DATA_BLOCK "ro_steam"   // DB283
{ S7_Optimized_Access := 'FALSE' }
VERSION : 0.1
// stored: InstanceOfName ro
"ro"
BEGIN
   P[1] := 0.1;
   P[2] := 0.2;
   P[3] := 0.3;
   P[4] := 0.4;
   P[5] := 0.5;
   P[6] := 0.6;
   P[7] := 0.7;
   P[8] := 0.8;
   P[9] := 0.9;
   P[10] := 1.0;
   T[1] := 10.0;
   T[2] := 20.0;
   T[3] := 30.0;
   T[4] := 40.0;
   T[5] := 50.0;
   T[6] := 60.0;
   T[7] := 70.0;
   T[8] := 80.0;
   T[9] := 90.0;
   T[10] := 100.0;
   T[11] := 110.0;
   T[12] := 120.0;
   T[13] := 130.0;
   T[14] := 140.0;
   T[15] := 150.0;
   T[16] := 160.0;
   T[17] := 170.0;
   T[18] := 180.0;
   T[19] := 190.0;
   T[20] := 200.0;
   PT[1,1] := 1.0003;
   PT[1,2] := 1.001799;
   PT[1,3] := 1.004368;
   PT[1,4] := 1.007838;
   PT[1,5] := 1.012099;
   PT[1,6] := 1.017078;
   PT[1,7] := 1.022727;
   PT[1,8] := 1.029017;
   PT[1,9] := 1.035929;
   PT[1,10] := 1729.941;
   PT[1,11] := 1779.703;
   PT[1,12] := 1829.026;
   PT[1,13] := 1878.016;
   PT[1,14] := 1926.736;
   PT[1,15] := 1975.238;
   PT[1,16] := 2023.559;
   PT[1,17] := 2071.728;
   PT[1,18] := 2119.771;
   PT[1,19] := 2167.707;
   PT[1,20] := 2215.552;
   PT[2,1] := 1.000253;
   PT[2,2] := 1.001754;
   PT[2,3] := 1.004324;
   PT[2,4] := 1.007794;
   PT[2,5] := 1.012055;
   PT[2,6] := 1.017033;
   PT[2,7] := 1.022682;
   PT[2,8] := 1.02897;
   PT[2,9] := 1.035881;
   PT[2,10] := 1.043407;
   PT[2,11] := 1.051552;
   PT[2,12] := 903.1196;
   PT[2,13] := 928.7784;
   PT[2,14] := 954.0966;
   PT[2,15] := 979.1605;
   PT[2,16] := 1004.021;
   PT[2,17] := 1028.715;
   PT[2,18] := 1053.271;
   PT[2,19] := 1077.71;
   PT[2,20] := 1102.051;
   PT[3,1] := 1.000206;
   PT[3,2] := 1.001709;
   PT[3,3] := 1.00428;
   PT[3,4] := 1.007751;
   PT[3,5] := 1.012011;
   PT[3,6] := 1.016989;
   PT[3,7] := 1.022637;
   PT[3,8] := 1.028924;
   PT[3,9] := 1.035833;
   PT[3,10] := 1.043357;
   PT[3,11] := 1.0515;
   PT[3,12] := 1.060273;
   PT[3,13] := 1.069697;
   PT[3,14] := 629.5558;
   PT[3,15] := 646.8893;
   PT[3,16] := 663.9833;
   PT[3,17] := 680.8912;
   PT[3,18] := 697.6475;
   PT[3,19] := 714.2781;
   PT[3,20] := 730.8032;
   PT[4,1] := 1.00016;
   PT[4,2] := 1.001664;
   PT[4,3] := 1.004236;
   PT[4,4] := 1.007707;
   PT[4,5] := 1.011968;
   PT[4,6] := 1.016945;
   PT[4,7] := 1.022592;
   PT[4,8] := 1.028878;
   PT[4,9] := 1.035785;
   PT[4,10] := 1.043307;
   PT[4,11] := 1.051447;
   PT[4,12] := 1.060218;
   PT[4,13] := 1.069639;
   PT[4,14] := 1.07974;
   PT[4,15] := 480.5462;
   PT[4,16] := 493.8126;
   PT[4,17] := 506.8611;
   PT[4,18] := 519.7418;
   PT[4,19] := 532.4865;
   PT[4,20] := 545.118;
   PT[5,1] := 1.000113;
   PT[5,2] := 1.001619;
   PT[5,3] := 1.004193;
   PT[5,4] := 1.007664;
   PT[5,5] := 1.011924;
   PT[5,6] := 1.016901;
   PT[5,7] := 1.022547;
   PT[5,8] := 1.028831;
   PT[5,9] := 1.035737;
   PT[5,10] := 1.043257;
   PT[5,11] := 1.051395;
   PT[5,12] := 1.060163;
   PT[5,13] := 1.06958;
   PT[5,14] := 1.079678;
   PT[5,15] := 1.090495;
   PT[5,16] := 391.5747;
   PT[5,17] := 402.3437;
   PT[5,18] := 412.9209;
   PT[5,19] := 423.3495;
   PT[5,20] := 433.6568;
   PT[6,1] := 1.000066;
   PT[6,2] := 1.001574;
   PT[6,3] := 1.004149;
   PT[6,4] := 1.00762;
   PT[6,5] := 1.01188;
   PT[6,6] := 1.016857;
   PT[6,7] := 1.022502;
   PT[6,8] := 1.028785;
   PT[6,9] := 1.035689;
   PT[6,10] := 1.043207;
   PT[6,11] := 1.051343;
   PT[6,12] := 1.060107;
   PT[6,13] := 1.069522;
   PT[6,14] := 1.079616;
   PT[6,15] := 1.090429;
   PT[6,16] := 323.2793;
   PT[6,17] := 332.5752;
   PT[6,18] := 341.6396;
   PT[6,19] := 350.5385;
   PT[6,20] := 359.3066;
   PT[7,1] := 1.000019;
   PT[7,2] := 1.001529;
   PT[7,3] := 1.004105;
   PT[7,4] := 1.007577;
   PT[7,5] := 1.011837;
   PT[7,6] := 1.016812;
   PT[7,7] := 1.022457;
   PT[7,8] := 1.028738;
   PT[7,9] := 1.035641;
   PT[7,10] := 1.043157;
   PT[7,11] := 1.05129;
   PT[7,12] := 1.060052;
   PT[7,13] := 1.069464;
   PT[7,14] := 1.079554;
   PT[7,15] := 1.090363;
   PT[7,16] := 1.101939;
   PT[7,17] := 282.652;
   PT[7,18] := 290.6629;
   PT[7,19] := 298.4836;
   PT[7,20] := 306.162;
   PT[8,1] := 0.9999723;
   PT[8,2] := 1.001484;
   PT[8,3] := 1.004061;
   PT[8,4] := 1.007533;
   PT[8,5] := 1.011793;
   PT[8,6] := 1.016768;
   PT[8,7] := 1.022411;
   PT[8,8] := 1.028692;
   PT[8,9] := 1.035593;
   PT[8,10] := 1.043107;
   PT[8,11] := 1.051238;
   PT[8,12] := 1.059997;
   PT[8,13] := 1.069406;
   PT[8,14] := 1.079492;
   PT[8,15] := 1.090296;
   PT[8,16] := 1.101868;
   PT[8,17] := 245.1154;
   PT[8,18] := 252.3714;
   PT[8,19] := 259.3993;
   PT[8,20] := 266.2699;
   PT[9,1] := 0.9999255;
   PT[9,2] := 1.001439;
   PT[9,3] := 1.004017;
   PT[9,4] := 1.00749;
   PT[9,5] := 1.011749;
   PT[9,6] := 1.016724;
   PT[9,7] := 1.022366;
   PT[9,8] := 1.028646;
   PT[9,9] := 1.035545;
   PT[9,10] := 1.043057;
   PT[9,11] := 1.051186;
   PT[9,12] := 1.059942;
   PT[9,13] := 1.069347;
   PT[9,14] := 1.07943;
   PT[9,15] := 1.09023;
   PT[9,16] := 1.101797;
   PT[9,17] := 1.114191;
   PT[9,18] := 222.5293;
   PT[9,19] := 228.9597;
   PT[9,20] := 235.2116;
   PT[10,1] := 0.9998788;
   PT[10,2] := 1.001394;
   PT[10,3] := 1.003973;
   PT[10,4] := 1.007446;
   PT[10,5] := 1.011706;
   PT[10,6] := 1.01668;
   PT[10,7] := 1.022321;
   PT[10,8] := 1.0286;
   PT[10,9] := 1.035497;
   PT[10,10] := 1.043007;
   PT[10,11] := 1.051134;
   PT[10,12] := 1.059887;
   PT[10,13] := 1.069289;
   PT[10,14] := 1.079368;
   PT[10,15] := 1.090164;
   PT[10,16] := 1.101725;
   PT[10,17] := 1.114115;
   PT[10,18] := 198.5921;
   PT[10,19] := 204.568;
   PT[10,20] := 210.3359;
END_DATA_BLOCK

DATA_BLOCK "Qs_gas"   // DB284
{ S7_Optimized_Access := 'FALSE' }
VERSION : 0.1
// stored: InstanceOfName Qs
"Qs"
BEGIN
   ro_c := 0.7024;
   Xa := 0.00642;
   Xy := 0.00217;
END_DATA_BLOCK

DATA_BLOCK "Q1_water"   // DB286
{ S7_Optimized_Access := 'FALSE' }
VERSION : 0.1
   VAR
      Calorie : Real := 8160.0;   // Калорийность
      KPD : Real := 0.89;   // КПД
      "E" : Real := 566.0;   // Энтальпия
      Value : Real;   // Расход воды
   END_VAR
BEGIN
END_DATA_BLOCK

// folder: Analog_out

DATA_BLOCK "DV_control_frequency"   // DB149
{ S7_Optimized_Access := 'FALSE' }
AUTHOR : Dmitriy_Petrov
VERSION : 0.1
// Задание для ПЧ ДВ
// stored: InstanceOfName WRITE_ANALOG_SIGNAL
"WRITE_ANALOG_SIGNAL"
BEGIN
   N_module := 14;
   N_chanel := 1;
   HL_control_signal_new := 50.0;
   HL_control_signal := 50.0;
END_DATA_BLOCK

DATA_BLOCK "DS_control_frequency"   // DB150
{ S7_Optimized_Access := 'FALSE' }
AUTHOR : Dmitriy_Petrov
VERSION : 0.1
// Задание для ПЧ ДС
// stored: InstanceOfName WRITE_ANALOG_SIGNAL
"WRITE_ANALOG_SIGNAL"
BEGIN
   N_module := 14;
   N_chanel := 2;
   HL_control_signal_new := 50.0;
   HL_control_signal := 50.0;
END_DATA_BLOCK

// folder: Analog_sensors

DATA_BLOCK "T_water_before_economizer"   // DB1
{ S7_Optimized_Access := 'FALSE' }
AUTHOR : Dmitriy_Petrov
VERSION : 0.1
// Температура питательной воды перед экономайзером (град С)
// stored: InstanceOfName READ_ANALOG_SENSOR
"READ_ANALOG_SENSOR"
BEGIN
   N_module := 1;
   N_chanel := 1;
   HL_sensor_new := 200.0;
   HL_sensor := 200.0;
END_DATA_BLOCK

DATA_BLOCK "T_water_after_economizer"   // DB2
{ S7_Optimized_Access := 'FALSE' }
AUTHOR : Dmitriy_Petrov
VERSION : 0.1
// Температура питательной воды после экономайзера (град С)
// stored: InstanceOfName READ_ANALOG_SENSOR
"READ_ANALOG_SENSOR"
BEGIN
   N_module := 1;
   N_chanel := 2;
   HL_sensor_new := 200.0;
   HL_sensor := 200.0;
END_DATA_BLOCK

DATA_BLOCK "dP_water_boiler"   // DB3
{ S7_Optimized_Access := 'FALSE' }
AUTHOR : Dmitriy_Petrov
VERSION : 0.1
// Перепад давления питательной воды на котел (кПа)
// stored: InstanceOfName READ_ANALOG_SENSOR
"READ_ANALOG_SENSOR"
BEGIN
   N_module := 1;
   N_chanel := 3;
   HL_sensor_new := 63.0;
   HL_sensor := 63.0;
END_DATA_BLOCK

DATA_BLOCK "P_water_before_regul"   // DB4
{ S7_Optimized_Access := 'FALSE' }
AUTHOR : Dmitriy_Petrov
VERSION : 0.1
// Давление питательной воды до регулятора (МПа)
// stored: InstanceOfName READ_ANALOG_SENSOR
"READ_ANALOG_SENSOR"
BEGIN
   N_module := 1;
   N_chanel := 4;
   HL_sensor_new := 25.0;
   HL_sensor := 25.0;
END_DATA_BLOCK

DATA_BLOCK "P_water_after_regul"   // DB5
{ S7_Optimized_Access := 'FALSE' }
AUTHOR : Dmitriy_Petrov
VERSION : 0.1
// Давление питательной воды после регулятора (МПа)
// stored: InstanceOfName READ_ANALOG_SENSOR
"READ_ANALOG_SENSOR"
BEGIN
   N_module := 1;
   N_chanel := 5;
   HL_sensor_new := 2.5;
   HL_sensor := 2.5;
END_DATA_BLOCK

DATA_BLOCK "dP_steam"   // DB6
{ S7_Optimized_Access := 'FALSE' }
AUTHOR : Dmitriy_Petrov
VERSION : 0.1
// Перепад давления пара в магистраль (кПа)
// stored: InstanceOfName READ_ANALOG_SENSOR
"READ_ANALOG_SENSOR"
BEGIN
   N_module := 1;
   N_chanel := 6;
END_DATA_BLOCK

DATA_BLOCK "P_steam"   // DB7
{ S7_Optimized_Access := 'FALSE' }
AUTHOR : Dmitriy_Petrov
VERSION : 0.1
// Давление пара в барабане (МПа)
// stored: InstanceOfName READ_ANALOG_SENSOR
"READ_ANALOG_SENSOR"
BEGIN
   N_module := 1;
   N_chanel := 7;
   HL_sensor_new := 16.0;
   HL_sensor := 16.0;
END_DATA_BLOCK

DATA_BLOCK "dP_furnace_boiler"   // DB8
{ S7_Optimized_Access := 'FALSE' }
AUTHOR : Dmitriy_Petrov
VERSION : 0.1
// Разрежение в топке котла (Па)
// stored: InstanceOfName READ_ANALOG_SENSOR
"READ_ANALOG_SENSOR"
BEGIN
   N_module := 2;
   N_chanel := 1;
   LL_sensor_new := -125.0;
   HL_sensor_new := 125.0;
   LL_sensor := -125.0;
   HL_sensor := 125.0;
END_DATA_BLOCK

DATA_BLOCK "P_gas_between_PZK1_and_PZK2"   // DB9
{ S7_Optimized_Access := 'FALSE' }
AUTHOR : Dmitriy_Petrov
VERSION : 0.1
// Давление газа между ПЗК-1 и ПЗК-2 (кПа)
// stored: InstanceOfName READ_ANALOG_SENSOR
"READ_ANALOG_SENSOR"
BEGIN
   HL_sensor_new := 63.0;
   HL_sensor := 63.0;
   N_module := 2;
   N_chanel := 2;
END_DATA_BLOCK

DATA_BLOCK "P_gas_before_burner"   // DB10
{ S7_Optimized_Access := 'FALSE' }
AUTHOR : Dmitriy_Petrov
VERSION : 0.1
// Давление газа перед горелкой (кПа)
// stored: InstanceOfName READ_ANALOG_SENSOR
"READ_ANALOG_SENSOR"
BEGIN
   N_module := 2;
   N_chanel := 3;
   HL_sensor_new := 40.0;
   HL_sensor := 40.0;
END_DATA_BLOCK

DATA_BLOCK "P_air_burner"   // DB11
{ S7_Optimized_Access := 'FALSE' }
AUTHOR : Dmitriy_Petrov
VERSION : 0.1
// Давление воздуха к горелке (Па)
// stored: InstanceOfName READ_ANALOG_SENSOR
"READ_ANALOG_SENSOR"
BEGIN
   N_module := 2;
   N_chanel := 4;
   HL_sensor_new := 2500.0;
   HL_sensor := 2500.0;
END_DATA_BLOCK

DATA_BLOCK "ZRW_position"   // DB12
{ S7_Optimized_Access := 'FALSE' }
AUTHOR : Dmitriy_Petrov
VERSION : 0.1
// Положение рег. заслонки питательной воды на котел (%)
// stored: InstanceOfName READ_ANALOG_SENSOR
"READ_ANALOG_SENSOR"
BEGIN
   N_module := 2;
   N_chanel := 5;
   LL_ADC_new := 8474;
   HL_ADC_new := 21888;
   LL_ADC := 8474;
   HL_ADC := 21888;
END_DATA_BLOCK

DATA_BLOCK "ZRG_position"   // DB13
{ S7_Optimized_Access := 'FALSE' }
AUTHOR : Dmitriy_Petrov
VERSION : 0.1
// Положение рег. заслонки газа перед котлом (%)
// stored: InstanceOfName READ_ANALOG_SENSOR
"READ_ANALOG_SENSOR"
BEGIN
   N_module := 2;
   N_chanel := 6;
   LL_ADC_new := 3056;
   HL_ADC_new := 25773;
   LL_ADC := 3056;
   HL_ADC := 25773;
END_DATA_BLOCK

DATA_BLOCK "NAV_position"   // DB14
{ S7_Optimized_Access := 'FALSE' }
AUTHOR : Dmitriy_Petrov
VERSION : 0.1
// Положение направл. аппарата вентилятора (%)
// stored: InstanceOfName READ_ANALOG_SENSOR
"READ_ANALOG_SENSOR"
BEGIN
   N_module := 2;
   N_chanel := 7;
   LL_ADC_new := 3658;
   HL_ADC_new := 26608;
   LL_ADC := 3658;
   HL_ADC := 26608;
END_DATA_BLOCK

DATA_BLOCK "NAD_position"   // DB15
{ S7_Optimized_Access := 'FALSE' }
AUTHOR : Dmitriy_Petrov
VERSION : 0.1
// Положение направл. аппарата дымососа (%)
// stored: InstanceOfName READ_ANALOG_SENSOR
"READ_ANALOG_SENSOR"
BEGIN
   N_module := 2;
   N_chanel := 8;
   LL_ADC_new := 2066;
   LL_ADC := 2066;
   HL_ADC_new := 24982;
   HL_ADC := 24982;
END_DATA_BLOCK

DATA_BLOCK "T_exhaust_gas_before_economizer"   // DB16
{ S7_Optimized_Access := 'FALSE' }
AUTHOR : Dmitriy_Petrov
VERSION : 0.1
// Температура уходящих дымовых газов  перед экономайзером (град С)
// stored: InstanceOfName READ_ANALOG_SENSOR
"READ_ANALOG_SENSOR"
BEGIN
   N_module := 3;
   N_chanel := 1;
   HL_sensor_new := 300.0;
   HL_sensor := 300.0;
END_DATA_BLOCK

DATA_BLOCK "T_exhaust_gas_after_economizer"   // DB17
{ S7_Optimized_Access := 'FALSE' }
AUTHOR : Dmitriy_Petrov
VERSION : 0.1
// Температура уходящих дымовых газов  после экономайзера (град С)
// stored: InstanceOfName READ_ANALOG_SENSOR
"READ_ANALOG_SENSOR"
BEGIN
   N_module := 3;
   N_chanel := 2;
   HL_sensor_new := 300.0;
   HL_sensor := 300.0;
END_DATA_BLOCK

DATA_BLOCK "dP_exhaust_gas_before_economizer"   // DB18
{ S7_Optimized_Access := 'FALSE' }
AUTHOR : Dmitriy_Petrov
VERSION : 0.1
// Разрежение в дымоходе перед экономайзером (Па)
// stored: InstanceOfName READ_ANALOG_SENSOR
"READ_ANALOG_SENSOR"
BEGIN
   N_module := 3;
   N_chanel := 3;
   LL_sensor_new := -2500.0;
   HL_sensor_new := 2500.0;
   LL_sensor := -2500.0;
   HL_sensor := 2500.0;
END_DATA_BLOCK

DATA_BLOCK "dP_exhaust_gas_after_economizer"   // DB19
{ S7_Optimized_Access := 'FALSE' }
AUTHOR : Dmitriy_Petrov
VERSION : 0.1
// Разрежение в дымоходе после экономайзера (Па)
// stored: InstanceOfName READ_ANALOG_SENSOR
"READ_ANALOG_SENSOR"
BEGIN
   N_module := 3;
   N_chanel := 4;
   LL_sensor_new := -2500.0;
   HL_sensor_new := 2500.0;
   LL_sensor := -2500.0;
   HL_sensor := 2500.0;
END_DATA_BLOCK

DATA_BLOCK "L_water"   // DB20
{ S7_Optimized_Access := 'FALSE' }
AUTHOR : Dmitriy_Petrov
VERSION : 0.1
// Уровень воды в барабане (мм)
// stored: InstanceOfName READ_ANALOG_SENSOR
"READ_ANALOG_SENSOR"
BEGIN
   N_module := 3;
   N_chanel := 5;
   LL_sensor_new := -315.0;
   HL_sensor_new := 315.0;
   LL_sensor := -315.0;
   HL_sensor := 315.0;
   LL_ADC_new := 27648;
   HL_ADC_new := 0;
   LL_ADC := 27648;
   HL_ADC := 0;
END_DATA_BLOCK

DATA_BLOCK "P_gas_before_BG"   // DB21
{ S7_Optimized_Access := 'FALSE' }
AUTHOR : Dmitriy_Petrov
VERSION : 0.1
// Давление газа перед БГ (кПа)
// stored: InstanceOfName READ_ANALOG_SENSOR
"READ_ANALOG_SENSOR"
BEGIN
   N_module := 3;
   N_chanel := 6;
   HL_sensor_new := 63.0;
   HL_sensor := 63.0;
END_DATA_BLOCK

DATA_BLOCK "T_gas_before_BG"   // DB22
{ S7_Optimized_Access := 'FALSE' }
AUTHOR : Dmitriy_Petrov
VERSION : 0.1
// Температура газа перед БГ (град С)
// stored: InstanceOfName READ_ANALOG_SENSOR
"READ_ANALOG_SENSOR"
BEGIN
   N_module := 3;
   N_chanel := 7;
   LL_sensor_new := -50.0;
   HL_sensor_new := 50.0;
   LL_sensor := -50.0;
   HL_sensor := 50.0;
END_DATA_BLOCK

DATA_BLOCK "P_steam_pipe"   // DB23
{ S7_Optimized_Access := 'FALSE' }
AUTHOR : Dmitriy_Petrov
VERSION : 0.1
// Давление пара в магистраль (МПа)
// stored: InstanceOfName READ_ANALOG_SENSOR
"READ_ANALOG_SENSOR"
BEGIN
   N_module := 3;
   N_chanel := 8;
   HL_sensor_new := 16.0;
   HL_sensor := 16.0;
END_DATA_BLOCK

DATA_BLOCK "T_steam"   // DB24
{ S7_Optimized_Access := 'FALSE' }
AUTHOR : Dmitriy_Petrov
VERSION : 0.1
// Температура пара в магистраль (град С)
// stored: InstanceOfName READ_ANALOG_SENSOR
"READ_ANALOG_SENSOR"
BEGIN
   N_module := 4;
   N_chanel := 1;
   HL_sensor_new := 300.0;
   HL_sensor := 300.0;
END_DATA_BLOCK

DATA_BLOCK "DV_current_frequency"   // DB25
{ S7_Optimized_Access := 'FALSE' }
AUTHOR : Dmitriy_Petrov
VERSION : 0.1
// Текущее значение частоты ПЧ вентилятора (Гц)
// stored: InstanceOfName READ_ANALOG_SENSOR
"READ_ANALOG_SENSOR"
BEGIN
   N_module := 4;
   N_chanel := 2;
   HL_sensor_new := 50.0;
   HL_sensor := 50.0;
END_DATA_BLOCK

DATA_BLOCK "DS_current_frequency"   // DB26
{ S7_Optimized_Access := 'FALSE' }
AUTHOR : Dmitriy_Petrov
VERSION : 0.1
// Текущее значение частоты ПЧ дымососа (Гц)
// stored: InstanceOfName READ_ANALOG_SENSOR
"READ_ANALOG_SENSOR"
BEGIN
   N_module := 4;
   N_chanel := 3;
   HL_sensor_new := 50.0;
   HL_sensor := 50.0;
END_DATA_BLOCK

DATA_BLOCK "Syst"   // DB243
{ S7_Optimized_Access := 'FALSE' }
VERSION : 0.1
   VAR
      First_scan_reg_map : Bool := true;
      Gen_imp : Bool;
   END_VAR
BEGIN
END_DATA_BLOCK

DATA_BLOCK "dP_water_level"   // DB287
{ S7_Optimized_Access := 'FALSE' }
AUTHOR : Dmitriy_Petrov
VERSION : 0.1
// stored: InstanceOfName READ_ANALOG_SENSOR
"READ_ANALOG_SENSOR"
BEGIN
   LL_ADC_new := 27648;
   HL_ADC_new := 0;
   LL_ADC := 27648;
   HL_ADC := 0;
   N_module := 3;
   N_chanel := 5;
END_DATA_BLOCK

DATA_BLOCK "L_water_level"   // DB288
{ S7_Optimized_Access := 'FALSE' }
AUTHOR : Dmitriy_Petrov
VERSION : 0.1
// stored: InstanceOfName READ_ANALOG_SENSOR
"READ_ANALOG_SENSOR"
BEGIN
   LL_sensor_new := -315.0;
   HL_sensor_new := 315.0;
   LL_ADC_new := 27648;
   HL_ADC_new := 0;
   N_module := 3;
   N_chanel := 5;
   LL_sensor := -315.0;
   HL_sensor := 315.0;
   LL_ADC := 27648;
   HL_ADC := 0;
END_DATA_BLOCK

// folder: Control

DATA_BLOCK "Control_ZRW"   // DB225
{ S7_Optimized_Access := 'FALSE' }
VERSION : 0.1
   VAR
      Mode : Bool;   // Режим управления (0-ручной, 1-автоматический)
      Manual_open : Bool;   // Ручное управление. Открыть
      Manual_close : Bool;   // Ручное управление. Закрыть
      Mode_from_PLC : Bool;   // Режим управления от ПЛК(0-ручной, 1-автоматический)
      Manual_open_from_PLC : Bool;   // Ручное управление от ПЛК. Открыть
      Manual_close_from_PLC : Bool;   // Ручное управление от ПЛК. Закрыть
      SP_PID : Real := 50.0;   // ПИД. Уставка
      DB_PID : Real := 4.0;   // ПИД. Зона нечувствительности
      KP_PID : Real := 0.4;   // ПИД. Кп
      TI_PID : UDInt := 30000;   // ПИД. Ти
      TD_PID : UDInt := 100;   // ПИД. Тд
      FMT_PID : UDInt := 30000;   // ПИД. Время хода исполнительного механизма (мс)
      DT_MIN_PID : UDInt := 200;   // ПИД. Величина минимальной длительности импульса (мс)
      GAP : DInt;   // ПИД. Люфт
   END_VAR
BEGIN
END_DATA_BLOCK

DATA_BLOCK "Control_ZRG"   // DB226
{ S7_Optimized_Access := 'FALSE' }
VERSION : 0.1
   VAR
      Mode : Bool;   // Режим управления (0-ручной, 1-автоматический)
      Manual_open : Bool;   // Ручное управление. Открыть
      Manual_close : Bool;   // Ручное управление. Закрыть
      Mode_from_PLC : Bool;   // Режим управления от ПЛК(0-ручной, 1-автоматический)
      Manual_open_from_PLC : Bool;   // Ручное управление от ПЛК. Открыть
      Manual_close_from_PLC : Bool;   // Ручное управление от ПЛК. Закрыть
      SP_PID : Real := 7.0;   // ПИД. Уставка
      DB_PID : Real := 0.1;   // ПИД. Зона нечувствительности
      KP_PID : Real := 0.4;   // ПИД. Кп
      TI_PID : UDInt := 3000;   // ПИД. Ти
      TD_PID : UDInt := 100;   // ПИД. Тд
      FMT_PID : UDInt := 30000;   // ПИД. Время хода исполнительного механизма (мс)
      DT_MIN_PID : UDInt := 150;   // ПИД. Величина минимальной длительности импульса (мс)
      GAP : DInt;   // ПИД. Люфт
   END_VAR
BEGIN
END_DATA_BLOCK

DATA_BLOCK "Control_ZDG"   // DB227
{ S7_Optimized_Access := 'FALSE' }
VERSION : 0.1
   VAR
      Mode : Bool;   // Режим управления (0-ручной, 1-автоматический)
      Manual_open : Bool;   // Ручное управление. Открыть
      Manual_close : Bool;   // Ручное управление. Закрыть
      Manual_stop : Bool;   // Ручное управление. Стоп
      Avto_open : Bool;   // Автоматическое управление. Открыть
      Avto_close : Bool;   // Автоматическое управление. Закрыть
      Avto_stop : Bool;   // Автоматическое управление. Стоп
   END_VAR
BEGIN
END_DATA_BLOCK

DATA_BLOCK "Control_GPZ"   // DB228
{ S7_Optimized_Access := 'FALSE' }
VERSION : 0.1
   VAR
      Mode : Bool;   // Режим управления (0-ручной, 1-автоматический)
      Manual_open : Bool;   // Ручное управление. Открыть
      Manual_close : Bool;   // Ручное управление. Закрыть
      Manual_stop : Bool;   // Ручное управление. Стоп
      Avto_open : Bool;   // Автоматическое управление. Открыть
      Avto_close : Bool;   // Автоматическое управление. Закрыть
      Avto_stop : Bool;   // Автоматическое управление. Стоп
   END_VAR
BEGIN
END_DATA_BLOCK

DATA_BLOCK "Control_KB"   // DB229
{ S7_Optimized_Access := 'FALSE' }
VERSION : 0.1
   VAR
      Mode : Bool;   // Режим управления (0-ручной, 1-автоматический)
      Manual_close : Bool;   // Ручное управление. Закрыть
      Avto_close : Bool;   // Автоматическое управление. Закрыть
   END_VAR
BEGIN
END_DATA_BLOCK

DATA_BLOCK "Control_KO"   // DB230
{ S7_Optimized_Access := 'FALSE' }
VERSION : 0.1
   VAR
      Mode : Bool;   // Режим управления (0-ручной, 1-автоматический)
      Manual_open : Bool;   // Ручное управление. Открыть
      Avto_open : Bool;   // Автоматическое управление. Открыть
   END_VAR
BEGIN
END_DATA_BLOCK

DATA_BLOCK "Control_KZ"   // DB231
{ S7_Optimized_Access := 'FALSE' }
VERSION : 0.1
   VAR
      Mode : Bool;   // Режим управления (0-ручной, 1-автоматический)
      Manual_open : Bool;   // Ручное управление. Открыть
      Avto_open : Bool;   // Автоматическое управление. Открыть
   END_VAR
BEGIN
END_DATA_BLOCK

DATA_BLOCK "Control_PZK1"   // DB232
{ S7_Optimized_Access := 'FALSE' }
VERSION : 0.1
   VAR
      Mode : Bool;   // Режим управления (0-ручной, 1-автоматический)
      Manual_open : Bool;   // Ручное управление. Открыть
      Avto_open : Bool;   // Автоматическое управление. Открыть
   END_VAR
BEGIN
END_DATA_BLOCK

DATA_BLOCK "Control_PZK2"   // DB233
{ S7_Optimized_Access := 'FALSE' }
VERSION : 0.1
   VAR
      Mode : Bool;   // Режим управления (0-ручной, 1-автоматический)
      Manual_open : Bool;   // Ручное управление. Открыть
      Avto_open : Bool;   // Автоматическое управление. Открыть
   END_VAR
BEGIN
END_DATA_BLOCK

DATA_BLOCK "Control_IVN"   // DB234
{ S7_Optimized_Access := 'FALSE' }
VERSION : 0.1
   VAR
      Mode : Bool;   // Режим управления (0-ручной, 1-автоматический)
      Manual_on : Bool;   // Ручное управление. Включить
      Avto_on : Bool;   // Автоматическое управление. Включить
   END_VAR
BEGIN
END_DATA_BLOCK

DATA_BLOCK "Control_ZDSV_before_boiler"   // DB235
{ S7_Optimized_Access := 'FALSE' }
VERSION : 0.1
   VAR
      Mode : Bool;   // Режим управления (0-ручной, 1-автоматический)
      Manual_open : Bool;   // Ручное управление. Открыть
      Manual_close : Bool;   // Ручное управление. Закрыть
      Manual_stop : Bool;   // Ручное управление. Стоп
      Avto_open : Bool;   // Автоматическое управление. Открыть
      Avto_close : Bool;   // Автоматическое управление. Закрыть
      Avto_stop : Bool;   // Автоматическое управление. Стоп
   END_VAR
BEGIN
END_DATA_BLOCK

DATA_BLOCK "Control_NAV"   // DB236
{ S7_Optimized_Access := 'FALSE' }
VERSION : 0.1
   VAR
      Mode : Bool;   // Режим управления (0-ручной, 1-автоматический)
      Manual_open : Bool;   // Ручное управление. Открыть
      Manual_close : Bool;   // Ручное управление. Закрыть
      Mode_from_PLC : Bool;   // Режим управления от ПЛК(0-ручной, 1-автоматический)
      Manual_open_from_PLC : Bool;   // Ручное управление от ПЛК. Открыть
      Manual_close_from_PLC : Bool;   // Ручное управление от ПЛК. Закрыть
      SP_PID : Real;   // ПИД. Уставка
      DB_PID : Real := 0.5;   // ПИД. Зона нечувствительности
      KP_PID : Real := 0.18;   // ПИД. Кп
      TI_PID : UDInt := 4769;   // ПИД. Ти
      TD_PID : UDInt := 0;   // ПИД. Тд
      FMT_PID : UDInt := 30000;   // ПИД. Время хода исполнительного механизма (мс)
      DT_MIN_PID : UDInt := 127;   // ПИД. Величина минимальной длительности импульса (мс)
      GAP : DInt;   // ПИД. Люфт
   END_VAR
BEGIN
END_DATA_BLOCK

DATA_BLOCK "Control_NAD"   // DB237
{ S7_Optimized_Access := 'FALSE' }
VERSION : 0.1
   VAR
      Mode : Bool;   // Режим управления (0-ручной, 1-автоматический)
      Manual_open : Bool;   // Ручное управление. Открыть
      Manual_close : Bool;   // Ручное управление. Закрыть
      Mode_from_PLC : Bool;   // Режим управления от ПЛК(0-ручной, 1-автоматический)
      Manual_open_from_PLC : Bool;   // Ручное управление от ПЛК. Открыть
      Manual_close_from_PLC : Bool;   // Ручное управление от ПЛК. Закрыть
      SP_PID : Real;   // ПИД. Уставка
      DB_PID : Real := 0.2;   // ПИД. Зона нечувствительности
      KP_PID : Real := 0.18;   // ПИД. Кп
      TI_PID : UDInt := 4891;   // ПИД. Ти
      TD_PID : UDInt := 0;   // ПИД. Тд
      FMT_PID : UDInt := 33000;   // ПИД. Время хода исполнительного механизма (мс)
      DT_MIN_PID : UDInt := 172;   // ПИД. Величина минимальной длительности импульса (мс)
      GAP : DInt;   // ПИД. Люфт
   END_VAR
BEGIN
END_DATA_BLOCK

DATA_BLOCK "Control_DV"   // DB238
{ S7_Optimized_Access := 'FALSE' }
VERSION : 0.1
   VAR
      Mode : Bool;   // Режим управления (0-ручной, 1-автоматический)
      Manual_Start : Bool;   // Ручное управление. Пуск
      Manual_Stop : Bool;   // Ручное управление. Стоп
      Manual_frequency : Real;   // Ручное управление. Задание частоты
      Avto_Start : Bool;   // Автоматическое управление. Пуск
      Avto_Stop : Bool;   // Автоматическое управление. Стоп
      Mode_from_PLC : Bool;   // Режим управления от ПЛК(0-ручной, 1-автоматический)
      Manual_frequency_from_PLC : Real;   // Ручное управление. Задание частоты
      SP_PID : Real;   // ПИД. Уставка
      DB_PID : Real := 10.0;   // ПИД. Зона нечувствительности
      KP_PID : Real := 0.05;   // ПИД. Кп
      TI_PID : UDInt := 10000;   // ПИД. Ти
      TD_PID : UDInt := 0;   // ПИД. Тд
   END_VAR
BEGIN
END_DATA_BLOCK

DATA_BLOCK "Control_DS"   // DB239
{ S7_Optimized_Access := 'FALSE' }
VERSION : 0.1
   VAR
      Mode : Bool;   // Режим управления (0-ручной, 1-автоматический)
      Manual_Start : Bool;   // Ручное управление. Пуск
      Manual_Stop : Bool;   // Ручное управление. Стоп
      Manual_frequency : Real;   // Ручное управление. Задание частоты
      Avto_Start : Bool;   // Автоматическое управление. Пуск
      Avto_Stop : Bool;   // Автоматическое управление. Стоп
      Mode_from_PLC : Bool;   // Режим управления от ПЛК(0-ручной, 1-автоматический)
      Manual_frequency_from_PLC : Real;   // Ручное управление. Задание частоты
      SP_PID : Real;   // ПИД. Уставка
      DB_PID : Real := 2.0;   // ПИД. Зона нечувствительности
      KP_PID : Real := 0.05;   // ПИД. Кп
      TI_PID : UDInt := 3000;   // ПИД. Ти
      TD_PID : UDInt := 0;   // ПИД. Тд
   END_VAR
BEGIN
END_DATA_BLOCK

// folder: Discrete_out

DATA_BLOCK "ZRG_control_open"   // DB114
{ S7_Optimized_Access := 'FALSE' }
AUTHOR : Dmitriy_Petrov
VERSION : 0.1
// ЗРГ Команда «Больше»
// stored: InstanceOfName WRITE_DISCRET_SIGNAL
"WRITE_DISCRET_SIGNAL"
BEGIN
   N_module := 11;
   N_chanel := 1;
END_DATA_BLOCK

DATA_BLOCK "ZRG_control_close"   // DB115
{ S7_Optimized_Access := 'FALSE' }
AUTHOR : Dmitriy_Petrov
VERSION : 0.1
// ЗРГ Команда «Меньше»
// stored: InstanceOfName WRITE_DISCRET_SIGNAL
"WRITE_DISCRET_SIGNAL"
BEGIN
   N_module := 11;
   N_chanel := 2;
END_DATA_BLOCK

DATA_BLOCK "NAV_control_open"   // DB116
{ S7_Optimized_Access := 'FALSE' }
AUTHOR : Dmitriy_Petrov
VERSION : 0.1
// НАВ Команда «Больше»
// stored: InstanceOfName WRITE_DISCRET_SIGNAL
"WRITE_DISCRET_SIGNAL"
BEGIN
   N_module := 11;
   N_chanel := 3;
END_DATA_BLOCK

DATA_BLOCK "NAV_control_close"   // DB117
{ S7_Optimized_Access := 'FALSE' }
AUTHOR : Dmitriy_Petrov
VERSION : 0.1
// НАВ Команда «Меньше»
// stored: InstanceOfName WRITE_DISCRET_SIGNAL
"WRITE_DISCRET_SIGNAL"
BEGIN
   N_module := 11;
   N_chanel := 4;
END_DATA_BLOCK

DATA_BLOCK "NAD_control_open"   // DB118
{ S7_Optimized_Access := 'FALSE' }
AUTHOR : Dmitriy_Petrov
VERSION : 0.1
// НАД Команда «Больше»
// stored: InstanceOfName WRITE_DISCRET_SIGNAL
"WRITE_DISCRET_SIGNAL"
BEGIN
   N_module := 11;
   N_chanel := 5;
END_DATA_BLOCK

DATA_BLOCK "NAD_control_close"   // DB119
{ S7_Optimized_Access := 'FALSE' }
AUTHOR : Dmitriy_Petrov
VERSION : 0.1
// НАД Команда «Меньше»
// stored: InstanceOfName WRITE_DISCRET_SIGNAL
"WRITE_DISCRET_SIGNAL"
BEGIN
   N_module := 11;
   N_chanel := 6;
END_DATA_BLOCK

DATA_BLOCK "ZRW_control_open"   // DB120
{ S7_Optimized_Access := 'FALSE' }
AUTHOR : Dmitriy_Petrov
VERSION : 0.1
// ЗРВ Команда «Больше»
// stored: InstanceOfName WRITE_DISCRET_SIGNAL
"WRITE_DISCRET_SIGNAL"
BEGIN
   N_module := 11;
   N_chanel := 7;
END_DATA_BLOCK

DATA_BLOCK "ZRW_control_close"   // DB121
{ S7_Optimized_Access := 'FALSE' }
AUTHOR : Dmitriy_Petrov
VERSION : 0.1
// ЗРВ Команда «Меньше»
// stored: InstanceOfName WRITE_DISCRET_SIGNAL
"WRITE_DISCRET_SIGNAL"
BEGIN
   N_module := 11;
   N_chanel := 8;
END_DATA_BLOCK

DATA_BLOCK "Indication_RUN"   // DB122
{ S7_Optimized_Access := 'FALSE' }
AUTHOR : Dmitriy_Petrov
VERSION : 0.1
// Индикация «Работа»
// stored: InstanceOfName WRITE_DISCRET_SIGNAL
"WRITE_DISCRET_SIGNAL"
BEGIN
   N_module := 11;
   N_chanel := 9;
END_DATA_BLOCK

DATA_BLOCK "Indication_ALARM"   // DB123
{ S7_Optimized_Access := 'FALSE' }
AUTHOR : Dmitriy_Petrov
VERSION : 0.1
// Индикация «Авария»
// stored: InstanceOfName WRITE_DISCRET_SIGNAL
"WRITE_DISCRET_SIGNAL"
BEGIN
   N_module := 11;
   N_chanel := 10;
END_DATA_BLOCK

DATA_BLOCK "Indication_NORMA"   // DB124
{ S7_Optimized_Access := 'FALSE' }
AUTHOR : Dmitriy_Petrov
VERSION : 0.1
// Индикация «Защиты в норме»
// stored: InstanceOfName WRITE_DISCRET_SIGNAL
"WRITE_DISCRET_SIGNAL"
BEGIN
   N_module := 11;
   N_chanel := 11;
END_DATA_BLOCK

DATA_BLOCK "Indication_READY"   // DB125
{ S7_Optimized_Access := 'FALSE' }
AUTHOR : Dmitriy_Petrov
VERSION : 0.1
// Индикация «Готов к розжигу»
// stored: InstanceOfName WRITE_DISCRET_SIGNAL
"WRITE_DISCRET_SIGNAL"
BEGIN
   N_module := 11;
   N_chanel := 12;
END_DATA_BLOCK

DATA_BLOCK "ZDG_control_open"   // DB126
{ S7_Optimized_Access := 'FALSE' }
AUTHOR : Dmitriy_Petrov
VERSION : 0.1
// ЗДГ команда «открыть»
// stored: InstanceOfName WRITE_DISCRET_SIGNAL
"WRITE_DISCRET_SIGNAL"
BEGIN
   N_module := 12;
   N_chanel := 1;
END_DATA_BLOCK

DATA_BLOCK "ZDG_control_close"   // DB127
{ S7_Optimized_Access := 'FALSE' }
AUTHOR : Dmitriy_Petrov
VERSION : 0.1
// ЗДГ команда «закрыть»
// stored: InstanceOfName WRITE_DISCRET_SIGNAL
"WRITE_DISCRET_SIGNAL"
BEGIN
   N_module := 12;
   N_chanel := 2;
END_DATA_BLOCK

DATA_BLOCK "ZDG_control_stop"   // DB128
{ S7_Optimized_Access := 'FALSE' }
AUTHOR : Dmitriy_Petrov
VERSION : 0.1
// ЗДГ команда «стоп»
// stored: InstanceOfName WRITE_DISCRET_SIGNAL
"WRITE_DISCRET_SIGNAL"
BEGIN
   N_module := 12;
   N_chanel := 3;
END_DATA_BLOCK

DATA_BLOCK "ZDG_control_disable_open"   // DB129
{ S7_Optimized_Access := 'FALSE' }
AUTHOR : Dmitriy_Petrov
VERSION : 0.1
// ЗДГ команда «запрет открытия»
// stored: InstanceOfName WRITE_DISCRET_SIGNAL
"WRITE_DISCRET_SIGNAL"
BEGIN
   N_module := 12;
   N_chanel := 4;
END_DATA_BLOCK

DATA_BLOCK "KB_control_close"   // DB130
{ S7_Optimized_Access := 'FALSE' }
AUTHOR : Dmitriy_Petrov
VERSION : 0.1
// КБ команда «закрыть»
// stored: InstanceOfName WRITE_DISCRET_SIGNAL
"WRITE_DISCRET_SIGNAL"
BEGIN
   N_module := 12;
   N_chanel := 5;
END_DATA_BLOCK

DATA_BLOCK "KO_control_open"   // DB131
{ S7_Optimized_Access := 'FALSE' }
AUTHOR : Dmitriy_Petrov
VERSION : 0.1
// КО команда «открыть»
// stored: InstanceOfName WRITE_DISCRET_SIGNAL
"WRITE_DISCRET_SIGNAL"
BEGIN
   N_module := 12;
   N_chanel := 6;
END_DATA_BLOCK

DATA_BLOCK "KZ_control_open"   // DB132
{ S7_Optimized_Access := 'FALSE' }
AUTHOR : Dmitriy_Petrov
VERSION : 0.1
// КЗ команда «открыть»
// stored: InstanceOfName WRITE_DISCRET_SIGNAL
"WRITE_DISCRET_SIGNAL"
BEGIN
   N_module := 12;
   N_chanel := 7;
END_DATA_BLOCK

DATA_BLOCK "IVN_control_on"   // DB133
{ S7_Optimized_Access := 'FALSE' }
AUTHOR : Dmitriy_Petrov
VERSION : 0.1
// ИВН команда «включить»
// stored: InstanceOfName WRITE_DISCRET_SIGNAL
"WRITE_DISCRET_SIGNAL"
BEGIN
   N_module := 12;
   N_chanel := 8;
END_DATA_BLOCK

DATA_BLOCK "PZK1_control_open"   // DB134
{ S7_Optimized_Access := 'FALSE' }
AUTHOR : Dmitriy_Petrov
VERSION : 0.1
// ПЗК1 команда «открыть»
// stored: InstanceOfName WRITE_DISCRET_SIGNAL
"WRITE_DISCRET_SIGNAL"
BEGIN
   N_module := 12;
   N_chanel := 9;
END_DATA_BLOCK

DATA_BLOCK "PZK2_control_open"   // DB135
{ S7_Optimized_Access := 'FALSE' }
AUTHOR : Dmitriy_Petrov
VERSION : 0.1
// ПЗК2 команда «открыть»
// stored: InstanceOfName WRITE_DISCRET_SIGNAL
"WRITE_DISCRET_SIGNAL"
BEGIN
   N_module := 12;
   N_chanel := 10;
END_DATA_BLOCK

DATA_BLOCK "ZDSV_before_boiler_control_open"   // DB136
{ S7_Optimized_Access := 'FALSE' }
AUTHOR : Dmitriy_Petrov
VERSION : 0.1
// ЗДСВ перед котлом команда «открыть»
// stored: InstanceOfName WRITE_DISCRET_SIGNAL
"WRITE_DISCRET_SIGNAL"
BEGIN
   N_module := 12;
   N_chanel := 11;
END_DATA_BLOCK

DATA_BLOCK "ZDSV_before_boiler_control_close"   // DB137
{ S7_Optimized_Access := 'FALSE' }
AUTHOR : Dmitriy_Petrov
VERSION : 0.1
// ЗДСВ перед котлом команда «закрыть»
// stored: InstanceOfName WRITE_DISCRET_SIGNAL
"WRITE_DISCRET_SIGNAL"
BEGIN
   N_module := 12;
   N_chanel := 12;
END_DATA_BLOCK

DATA_BLOCK "ZDSV_before_boiler_control_stop"   // DB138
{ S7_Optimized_Access := 'FALSE' }
AUTHOR : Dmitriy_Petrov
VERSION : 0.1
// ЗДСВ перед котлом команда «стоп»
// stored: InstanceOfName WRITE_DISCRET_SIGNAL
"WRITE_DISCRET_SIGNAL"
BEGIN
   N_module := 12;
   N_chanel := 13;
END_DATA_BLOCK

DATA_BLOCK "ZDSV_before_boiler_control_disable_close"   // DB139
{ S7_Optimized_Access := 'FALSE' }
AUTHOR : Dmitriy_Petrov
VERSION : 0.1
// ЗДСВ перед котлом команда «разрешение на закрытие»
// stored: InstanceOfName WRITE_DISCRET_SIGNAL
"WRITE_DISCRET_SIGNAL"
BEGIN
   N_module := 12;
   N_chanel := 14;
END_DATA_BLOCK

DATA_BLOCK "GPZ_control_open"   // DB140
{ S7_Optimized_Access := 'FALSE' }
AUTHOR : Dmitriy_Petrov
VERSION : 0.1
// ГПЗ команда «открыть»
// stored: InstanceOfName WRITE_DISCRET_SIGNAL
"WRITE_DISCRET_SIGNAL"
BEGIN
   N_module := 12;
   N_chanel := 15;
END_DATA_BLOCK

DATA_BLOCK "GPZ_control_close"   // DB141
{ S7_Optimized_Access := 'FALSE' }
AUTHOR : Dmitriy_Petrov
VERSION : 0.1
// ГПЗ команда «закрыть»
// stored: InstanceOfName WRITE_DISCRET_SIGNAL
"WRITE_DISCRET_SIGNAL"
BEGIN
   N_module := 12;
   N_chanel := 16;
END_DATA_BLOCK

DATA_BLOCK "GPZ_control_stop"   // DB142
{ S7_Optimized_Access := 'FALSE' }
AUTHOR : Dmitriy_Petrov
VERSION : 0.1
// ГПЗ команда «стоп»
// stored: InstanceOfName WRITE_DISCRET_SIGNAL
"WRITE_DISCRET_SIGNAL"
BEGIN
   N_module := 13;
   N_chanel := 1;
END_DATA_BLOCK

DATA_BLOCK "GPZ_control_disable_close"   // DB143
{ S7_Optimized_Access := 'FALSE' }
AUTHOR : Dmitriy_Petrov
VERSION : 0.1
// ГПЗ команда «разрешение на закрытие»
// stored: InstanceOfName WRITE_DISCRET_SIGNAL
"WRITE_DISCRET_SIGNAL"
BEGIN
   N_module := 13;
   N_chanel := 2;
END_DATA_BLOCK

DATA_BLOCK "control_alarm_signal"   // DB144
{ S7_Optimized_Access := 'FALSE' }
AUTHOR : Dmitriy_Petrov
VERSION : 0.1
// Включение аварийной сигнализации
// stored: InstanceOfName WRITE_DISCRET_SIGNAL
"WRITE_DISCRET_SIGNAL"
BEGIN
   N_module := 13;
   N_chanel := 3;
END_DATA_BLOCK

DATA_BLOCK "DV_control_start"   // DB145
{ S7_Optimized_Access := 'FALSE' }
AUTHOR : Dmitriy_Petrov
VERSION : 0.1
// ДВ команда «пуск»
// stored: InstanceOfName WRITE_DISCRET_SIGNAL
"WRITE_DISCRET_SIGNAL"
BEGIN
   N_module := 13;
   N_chanel := 4;
END_DATA_BLOCK

DATA_BLOCK "DV_control_stop"   // DB146
{ S7_Optimized_Access := 'FALSE' }
AUTHOR : Dmitriy_Petrov
VERSION : 0.1
// ДВ команда «стоп»
// stored: InstanceOfName WRITE_DISCRET_SIGNAL
"WRITE_DISCRET_SIGNAL"
BEGIN
   N_module := 13;
   N_chanel := 5;
END_DATA_BLOCK

DATA_BLOCK "DS_control_start"   // DB147
{ S7_Optimized_Access := 'FALSE' }
AUTHOR : Dmitriy_Petrov
VERSION : 0.1
// ДС команда «пуск»
// stored: InstanceOfName WRITE_DISCRET_SIGNAL
"WRITE_DISCRET_SIGNAL"
BEGIN
   N_module := 13;
   N_chanel := 6;
END_DATA_BLOCK

DATA_BLOCK "DS_control_stop"   // DB148
{ S7_Optimized_Access := 'FALSE' }
AUTHOR : Dmitriy_Petrov
VERSION : 0.1
// ДС команда «стоп»
// stored: InstanceOfName WRITE_DISCRET_SIGNAL
"WRITE_DISCRET_SIGNAL"
BEGIN
   N_module := 13;
   N_chanel := 7;
END_DATA_BLOCK

// folder: Discrete_sensors

DATA_BLOCK "Burner_flame"   // DB27
{ S7_Optimized_Access := 'FALSE' }
AUTHOR : Dmitriy_Petrov
VERSION : 0.1
// Наличие пламени горелки
// stored: InstanceOfName READ_DISCRET_SIGNAL
"READ_DISCRET_SIGNAL"
BEGIN
   N_module := 5;
   N_chanel := 1;
END_DATA_BLOCK

DATA_BLOCK "Igniter_flame"   // DB28
{ S7_Optimized_Access := 'FALSE' }
AUTHOR : Dmitriy_Petrov
VERSION : 0.1
// Наличие пламени запальника горелки
// stored: InstanceOfName READ_DISCRET_SIGNAL
"READ_DISCRET_SIGNAL"
BEGIN
   N_module := 5;
   N_chanel := 2;
END_DATA_BLOCK

DATA_BLOCK "KB_close"   // DB29
{ S7_Optimized_Access := 'FALSE' }
AUTHOR : Dmitriy_Petrov
VERSION : 0.1
// Клапан безопасности закрыт
// stored: InstanceOfName READ_DISCRET_SIGNAL
"READ_DISCRET_SIGNAL"
BEGIN
   N_module := 5;
   N_chanel := 3;
END_DATA_BLOCK

DATA_BLOCK "KO_open"   // DB30
{ S7_Optimized_Access := 'FALSE' }
AUTHOR : Dmitriy_Petrov
VERSION : 0.1
// Клапан опрессовки открыт
// stored: InstanceOfName READ_DISCRET_SIGNAL
"READ_DISCRET_SIGNAL"
BEGIN
   N_module := 5;
   N_chanel := 4;
END_DATA_BLOCK

DATA_BLOCK "KZ_open"   // DB31
{ S7_Optimized_Access := 'FALSE' }
AUTHOR : Dmitriy_Petrov
VERSION : 0.1
// Клапан запальника открыт
// stored: InstanceOfName READ_DISCRET_SIGNAL
"READ_DISCRET_SIGNAL"
BEGIN
   N_module := 5;
   N_chanel := 5;
END_DATA_BLOCK

DATA_BLOCK "PZK1_open"   // DB32
{ S7_Optimized_Access := 'FALSE' }
AUTHOR : Dmitriy_Petrov
VERSION : 0.1
// ПЗК-1 горелки открыт
// stored: InstanceOfName READ_DISCRET_SIGNAL
"READ_DISCRET_SIGNAL"
BEGIN
   N_module := 5;
   N_chanel := 6;
END_DATA_BLOCK

DATA_BLOCK "PZK2_not_close"   // DB33
{ S7_Optimized_Access := 'FALSE' }
AUTHOR : Dmitriy_Petrov
VERSION : 0.1
// ПЗК-2 горелки не закрыт
// stored: InstanceOfName READ_DISCRET_SIGNAL
"READ_DISCRET_SIGNAL"
BEGIN
   N_module := 5;
   N_chanel := 7;
   Enable := false;
END_DATA_BLOCK

DATA_BLOCK "P_gas_before_BG_min"   // DB34
{ S7_Optimized_Access := 'FALSE' }
AUTHOR : Dmitriy_Petrov
VERSION : 0.1
// Давление газа перед БГ мин.
// stored: InstanceOfName READ_DISCRET_SIGNAL
"READ_DISCRET_SIGNAL"
BEGIN
   N_module := 5;
   N_chanel := 8;
END_DATA_BLOCK

DATA_BLOCK "P_gas_before_BG_max"   // DB35
{ S7_Optimized_Access := 'FALSE' }
AUTHOR : Dmitriy_Petrov
VERSION : 0.1
// Давление газа перед БГ макс.
// stored: InstanceOfName READ_DISCRET_SIGNAL
"READ_DISCRET_SIGNAL"
BEGIN
   N_module := 5;
   N_chanel := 9;
END_DATA_BLOCK

DATA_BLOCK "P_air_before_burner_min"   // DB36
{ S7_Optimized_Access := 'FALSE' }
AUTHOR : Dmitriy_Petrov
VERSION : 0.1
// Давление воздуха перед горелкой мин.
// stored: InstanceOfName READ_DISCRET_SIGNAL
"READ_DISCRET_SIGNAL"
BEGIN
   N_module := 5;
   N_chanel := 10;
END_DATA_BLOCK

DATA_BLOCK "P_gas_before_burner_min"   // DB37
{ S7_Optimized_Access := 'FALSE' }
AUTHOR : Dmitriy_Petrov
VERSION : 0.1
// Давление газа перед горелкой мин.
// stored: InstanceOfName READ_DISCRET_SIGNAL
"READ_DISCRET_SIGNAL"
BEGIN
   N_module := 5;
   N_chanel := 11;
END_DATA_BLOCK

DATA_BLOCK "P_gas_before_burner_max"   // DB38
{ S7_Optimized_Access := 'FALSE' }
AUTHOR : Dmitriy_Petrov
VERSION : 0.1
// Давление газа перед горелкой макс.
// stored: InstanceOfName READ_DISCRET_SIGNAL
"READ_DISCRET_SIGNAL"
BEGIN
   N_module := 5;
   N_chanel := 12;
END_DATA_BLOCK

DATA_BLOCK "ZRG_open"   // DB39
{ S7_Optimized_Access := 'FALSE' }
AUTHOR : Dmitriy_Petrov
VERSION : 0.1
// Регулирующая заслонка газа открыта
// stored: InstanceOfName READ_DISCRET_SIGNAL
"READ_DISCRET_SIGNAL"
BEGIN
   N_module := 5;
   N_chanel := 13;
END_DATA_BLOCK

DATA_BLOCK "ZRG_close"   // DB40
{ S7_Optimized_Access := 'FALSE' }
AUTHOR : Dmitriy_Petrov
VERSION : 0.1
// Регулирующая заслонка газа закрыта
// stored: InstanceOfName READ_DISCRET_SIGNAL
"READ_DISCRET_SIGNAL"
BEGIN
   N_module := 5;
   N_chanel := 14;
END_DATA_BLOCK

DATA_BLOCK "ZRG_middle"   // DB41
{ S7_Optimized_Access := 'FALSE' }
AUTHOR : Dmitriy_Petrov
VERSION : 0.1
// Регулирующая заслонка газа среднее
// stored: InstanceOfName READ_DISCRET_SIGNAL
"READ_DISCRET_SIGNAL"
BEGIN
   N_module := 5;
   N_chanel := 15;
   Invert := true;
END_DATA_BLOCK

DATA_BLOCK "ZRG_avto"   // DB42
{ S7_Optimized_Access := 'FALSE' }
AUTHOR : Dmitriy_Petrov
VERSION : 0.1
// Регулирующая заслонка газа. БРУ в положении "Авт"
// stored: InstanceOfName READ_DISCRET_SIGNAL
"READ_DISCRET_SIGNAL"
BEGIN
   N_module := 5;
   N_chanel := 16;
END_DATA_BLOCK

DATA_BLOCK "NAV_open"   // DB43
{ S7_Optimized_Access := 'FALSE' }
AUTHOR : Dmitriy_Petrov
VERSION : 0.1
// НАВ открыт
// stored: InstanceOfName READ_DISCRET_SIGNAL
"READ_DISCRET_SIGNAL"
BEGIN
   N_module := 6;
   N_chanel := 1;
END_DATA_BLOCK

DATA_BLOCK "NAV_close"   // DB44
{ S7_Optimized_Access := 'FALSE' }
AUTHOR : Dmitriy_Petrov
VERSION : 0.1
// НАВ закрыт
// stored: InstanceOfName READ_DISCRET_SIGNAL
"READ_DISCRET_SIGNAL"
BEGIN
   N_module := 6;
   N_chanel := 2;
END_DATA_BLOCK

DATA_BLOCK "NAV_middle"   // DB45
{ S7_Optimized_Access := 'FALSE' }
AUTHOR : Dmitriy_Petrov
VERSION : 0.1
// НАВ среднее
// stored: InstanceOfName READ_DISCRET_SIGNAL
"READ_DISCRET_SIGNAL"
BEGIN
   N_module := 6;
   N_chanel := 3;
END_DATA_BLOCK

DATA_BLOCK "NAV_avto"   // DB46
{ S7_Optimized_Access := 'FALSE' }
AUTHOR : Dmitriy_Petrov
VERSION : 0.1
// НАВ. БРУ в положении "Авт"
// stored: InstanceOfName READ_DISCRET_SIGNAL
"READ_DISCRET_SIGNAL"
BEGIN
   N_module := 6;
   N_chanel := 4;
END_DATA_BLOCK

DATA_BLOCK "NAD_open"   // DB47
{ S7_Optimized_Access := 'FALSE' }
AUTHOR : Dmitriy_Petrov
VERSION : 0.1
// НАД открыт
// stored: InstanceOfName READ_DISCRET_SIGNAL
"READ_DISCRET_SIGNAL"
BEGIN
   N_module := 6;
   N_chanel := 5;
END_DATA_BLOCK

DATA_BLOCK "NAD_close"   // DB48
{ S7_Optimized_Access := 'FALSE' }
AUTHOR : Dmitriy_Petrov
VERSION : 0.1
// НАД закрыт
// stored: InstanceOfName READ_DISCRET_SIGNAL
"READ_DISCRET_SIGNAL"
BEGIN
   N_module := 6;
   N_chanel := 6;
END_DATA_BLOCK

DATA_BLOCK "NAD_middle"   // DB49
{ S7_Optimized_Access := 'FALSE' }
AUTHOR : Dmitriy_Petrov
VERSION : 0.1
// НАД среднее
// stored: InstanceOfName READ_DISCRET_SIGNAL
"READ_DISCRET_SIGNAL"
BEGIN
   N_module := 6;
   N_chanel := 7;
END_DATA_BLOCK

DATA_BLOCK "NAD_avto"   // DB50
{ S7_Optimized_Access := 'FALSE' }
AUTHOR : Dmitriy_Petrov
VERSION : 0.1
// НАД. БРУ в положении "Авт"
// stored: InstanceOfName READ_DISCRET_SIGNAL
"READ_DISCRET_SIGNAL"
BEGIN
   N_module := 6;
   N_chanel := 8;
END_DATA_BLOCK

DATA_BLOCK "PZK2_open"   // DB51
{ S7_Optimized_Access := 'FALSE' }
AUTHOR : Dmitriy_Petrov
VERSION : 0.1
// ПЗК-2 горелки открыт
// stored: InstanceOfName READ_DISCRET_SIGNAL
"READ_DISCRET_SIGNAL"
BEGIN
   N_module := 5;
   N_chanel := 7;
END_DATA_BLOCK

DATA_BLOCK "dP_furnace_boiler_min"   // DB52
{ S7_Optimized_Access := 'FALSE' }
AUTHOR : Dmitriy_Petrov
VERSION : 0.1
// Разрежение в топке котла мин.
// stored: InstanceOfName READ_DISCRET_SIGNAL
"READ_DISCRET_SIGNAL"
BEGIN
   N_module := 6;
   N_chanel := 10;
END_DATA_BLOCK

DATA_BLOCK "P_water_after_regul_min"   // DB53
{ S7_Optimized_Access := 'FALSE' }
AUTHOR : Dmitriy_Petrov
VERSION : 0.1
// Давление питательной воды после регулятора мин.
// stored: InstanceOfName READ_DISCRET_SIGNAL
"READ_DISCRET_SIGNAL"
BEGIN
   N_module := 6;
   N_chanel := 11;
END_DATA_BLOCK

DATA_BLOCK "P_steam_max"   // DB54
{ S7_Optimized_Access := 'FALSE' }
AUTHOR : Dmitriy_Petrov
VERSION : 0.1
// Давление пара в барабане макс.
// stored: InstanceOfName READ_DISCRET_SIGNAL
"READ_DISCRET_SIGNAL"
BEGIN
   N_module := 6;
   N_chanel := 12;
END_DATA_BLOCK

DATA_BLOCK "L_water_min"   // DB55
{ S7_Optimized_Access := 'FALSE' }
AUTHOR : Dmitriy_Petrov
VERSION : 0.1
// Уровень воды в барабане мин.
// stored: InstanceOfName READ_DISCRET_SIGNAL
"READ_DISCRET_SIGNAL"
BEGIN
   N_module := 6;
   N_chanel := 13;
END_DATA_BLOCK

DATA_BLOCK "L_water_max"   // DB56
{ S7_Optimized_Access := 'FALSE' }
AUTHOR : Dmitriy_Petrov
VERSION : 0.1
// Уровень воды в барабане макс.
// stored: InstanceOfName READ_DISCRET_SIGNAL
"READ_DISCRET_SIGNAL"
BEGIN
   N_module := 6;
   N_chanel := 14;
END_DATA_BLOCK

DATA_BLOCK "Call_power_supply_cabinet"   // DB57
{ S7_Optimized_Access := 'FALSE' }
AUTHOR : Dmitriy_Petrov
VERSION : 0.1
// Вызов к шкафу электропитания
// stored: InstanceOfName READ_DISCRET_SIGNAL
"READ_DISCRET_SIGNAL"
BEGIN
   N_module := 6;
   N_chanel := 15;
END_DATA_BLOCK

DATA_BLOCK "DV_Invertor_alarm"   // DB58
{ S7_Optimized_Access := 'FALSE' }
AUTHOR : Dmitriy_Petrov
VERSION : 0.1
// Авария ПЧ ДВ
// stored: InstanceOfName READ_DISCRET_SIGNAL
"READ_DISCRET_SIGNAL"
BEGIN
   N_module := 6;
   N_chanel := 16;
END_DATA_BLOCK

DATA_BLOCK "DV_local_control"   // DB59
{ S7_Optimized_Access := 'FALSE' }
AUTHOR : Dmitriy_Petrov
VERSION : 0.1
// Режим работы ДВ «Местный»
// stored: InstanceOfName READ_DISCRET_SIGNAL
"READ_DISCRET_SIGNAL"
BEGIN
   N_module := 7;
   N_chanel := 1;
END_DATA_BLOCK

DATA_BLOCK "DV_dist_control"   // DB60
{ S7_Optimized_Access := 'FALSE' }
AUTHOR : Dmitriy_Petrov
VERSION : 0.1
// Режим работы ДВ «Дистанционный»
// stored: InstanceOfName READ_DISCRET_SIGNAL
"READ_DISCRET_SIGNAL"
BEGIN
   N_module := 7;
   N_chanel := 2;
END_DATA_BLOCK

DATA_BLOCK "DV_powergrid_mode"   // DB61
{ S7_Optimized_Access := 'FALSE' }
AUTHOR : Dmitriy_Petrov
VERSION : 0.1
// Режим "СЕТЬ" ДВ
// stored: InstanceOfName READ_DISCRET_SIGNAL
"READ_DISCRET_SIGNAL"
BEGIN
   N_module := 7;
   N_chanel := 3;
END_DATA_BLOCK

DATA_BLOCK "DV_invertor_mode"   // DB62
{ S7_Optimized_Access := 'FALSE' }
AUTHOR : Dmitriy_Petrov
VERSION : 0.1
// Режим "ПЧ" ДВ
// stored: InstanceOfName READ_DISCRET_SIGNAL
"READ_DISCRET_SIGNAL"
BEGIN
   N_module := 7;
   N_chanel := 4;
END_DATA_BLOCK

DATA_BLOCK "DV_invertor_QF_on"   // DB63
{ S7_Optimized_Access := 'FALSE' }
AUTHOR : Dmitriy_Petrov
VERSION : 0.1
// Автомат работы ДВ от ПЧ включен
// stored: InstanceOfName READ_DISCRET_SIGNAL
"READ_DISCRET_SIGNAL"
BEGIN
   N_module := 7;
   N_chanel := 5;
END_DATA_BLOCK

DATA_BLOCK "DV_powergrid_QF_on"   // DB64
{ S7_Optimized_Access := 'FALSE' }
AUTHOR : Dmitriy_Petrov
VERSION : 0.1
// Автомат работы ДВ от сети включен
// stored: InstanceOfName READ_DISCRET_SIGNAL
"READ_DISCRET_SIGNAL"
BEGIN
   N_module := 7;
   N_chanel := 6;
END_DATA_BLOCK

DATA_BLOCK "DV_invertor_on"   // DB65
{ S7_Optimized_Access := 'FALSE' }
AUTHOR : Dmitriy_Petrov
VERSION : 0.1
// Включен ДВ от ПЧ
// stored: InstanceOfName READ_DISCRET_SIGNAL
"READ_DISCRET_SIGNAL"
BEGIN
   N_module := 7;
   N_chanel := 7;
END_DATA_BLOCK

DATA_BLOCK "DV_powergrid_on"   // DB66
{ S7_Optimized_Access := 'FALSE' }
AUTHOR : Dmitriy_Petrov
VERSION : 0.1
// Включен ДВ от сети
// stored: InstanceOfName READ_DISCRET_SIGNAL
"READ_DISCRET_SIGNAL"
BEGIN
   N_module := 7;
   N_chanel := 8;
END_DATA_BLOCK

DATA_BLOCK "DV_no_voltage"   // DB67
{ S7_Optimized_Access := 'FALSE' }
AUTHOR : Dmitriy_Petrov
VERSION : 0.1
// Нет напряжения сети ШУД ДВ
// stored: InstanceOfName READ_DISCRET_SIGNAL
"READ_DISCRET_SIGNAL"
BEGIN
   N_module := 7;
   N_chanel := 9;
   Invert := true;
END_DATA_BLOCK

DATA_BLOCK "DS_Invertor_alarm"   // DB68
{ S7_Optimized_Access := 'FALSE' }
AUTHOR : Dmitriy_Petrov
VERSION : 0.1
// Авария ПЧ ДС
// stored: InstanceOfName READ_DISCRET_SIGNAL
"READ_DISCRET_SIGNAL"
BEGIN
   N_module := 7;
   N_chanel := 10;
END_DATA_BLOCK

DATA_BLOCK "DS_local_control"   // DB69
{ S7_Optimized_Access := 'FALSE' }
AUTHOR : Dmitriy_Petrov
VERSION : 0.1
// Режим работы ДС «Местный»
// stored: InstanceOfName READ_DISCRET_SIGNAL
"READ_DISCRET_SIGNAL"
BEGIN
   N_module := 7;
   N_chanel := 11;
END_DATA_BLOCK

DATA_BLOCK "DS_dist_control"   // DB70
{ S7_Optimized_Access := 'FALSE' }
AUTHOR : Dmitriy_Petrov
VERSION : 0.1
// Режим работы ДC «Дистанционный»
// stored: InstanceOfName READ_DISCRET_SIGNAL
"READ_DISCRET_SIGNAL"
BEGIN
   N_module := 7;
   N_chanel := 12;
END_DATA_BLOCK

DATA_BLOCK "DS_powergrid_mode"   // DB71
{ S7_Optimized_Access := 'FALSE' }
AUTHOR : Dmitriy_Petrov
VERSION : 0.1
// Режим "СЕТЬ" ДC
// stored: InstanceOfName READ_DISCRET_SIGNAL
"READ_DISCRET_SIGNAL"
BEGIN
   N_module := 7;
   N_chanel := 13;
END_DATA_BLOCK

DATA_BLOCK "DS_invertor_mode"   // DB72
{ S7_Optimized_Access := 'FALSE' }
AUTHOR : Dmitriy_Petrov
VERSION : 0.1
// Режим "ПЧ" ДС
// stored: InstanceOfName READ_DISCRET_SIGNAL
"READ_DISCRET_SIGNAL"
BEGIN
   N_module := 7;
   N_chanel := 14;
END_DATA_BLOCK

DATA_BLOCK "DS_invertor_QF_on"   // DB73
{ S7_Optimized_Access := 'FALSE' }
AUTHOR : Dmitriy_Petrov
VERSION : 0.1
// Автомат работы ДС от ПЧ включен
// stored: InstanceOfName READ_DISCRET_SIGNAL
"READ_DISCRET_SIGNAL"
BEGIN
   N_module := 7;
   N_chanel := 15;
END_DATA_BLOCK

DATA_BLOCK "DS_powergrid_QF_on"   // DB74
{ S7_Optimized_Access := 'FALSE' }
AUTHOR : Dmitriy_Petrov
VERSION : 0.1
// Автомат работы ДС от сети включен
// stored: InstanceOfName READ_DISCRET_SIGNAL
"READ_DISCRET_SIGNAL"
BEGIN
   N_module := 7;
   N_chanel := 16;
END_DATA_BLOCK

DATA_BLOCK "DS_invertor_on"   // DB75
{ S7_Optimized_Access := 'FALSE' }
AUTHOR : Dmitriy_Petrov
VERSION : 0.1
// Включен ДС от ПЧ
// stored: InstanceOfName READ_DISCRET_SIGNAL
"READ_DISCRET_SIGNAL"
BEGIN
   N_module := 8;
   N_chanel := 1;
END_DATA_BLOCK

DATA_BLOCK "DS_powergrid_on"   // DB76
{ S7_Optimized_Access := 'FALSE' }
AUTHOR : Dmitriy_Petrov
VERSION : 0.1
// Включен ДС от сети
// stored: InstanceOfName READ_DISCRET_SIGNAL
"READ_DISCRET_SIGNAL"
BEGIN
   N_module := 8;
   N_chanel := 2;
END_DATA_BLOCK

DATA_BLOCK "DS_no_voltage"   // DB77
{ S7_Optimized_Access := 'FALSE' }
AUTHOR : Dmitriy_Petrov
VERSION : 0.1
// Нет напряжения сети ШУД ДС
// stored: InstanceOfName READ_DISCRET_SIGNAL
"READ_DISCRET_SIGNAL"
BEGIN
   N_module := 8;
   N_chanel := 3;
   Invert := true;
END_DATA_BLOCK

DATA_BLOCK "CO_1"   // DB78
{ S7_Optimized_Access := 'FALSE' }
AUTHOR : Dmitriy_Petrov
VERSION : 0.1
// Загазованность СО I порог
// stored: InstanceOfName READ_DISCRET_SIGNAL
"READ_DISCRET_SIGNAL"
BEGIN
   N_module := 8;
   N_chanel := 4;
END_DATA_BLOCK

DATA_BLOCK "CO_2"   // DB79
{ S7_Optimized_Access := 'FALSE' }
AUTHOR : Dmitriy_Petrov
VERSION : 0.1
// Загазованность СО II порог
// stored: InstanceOfName READ_DISCRET_SIGNAL
"READ_DISCRET_SIGNAL"
BEGIN
   N_module := 8;
   N_chanel := 5;
END_DATA_BLOCK

DATA_BLOCK "CH4"   // DB80
{ S7_Optimized_Access := 'FALSE' }
AUTHOR : Dmitriy_Petrov
VERSION : 0.1
// Загазованность CH4 порог
// stored: InstanceOfName READ_DISCRET_SIGNAL
"READ_DISCRET_SIGNAL"
BEGIN
   N_module := 8;
   N_chanel := 6;
END_DATA_BLOCK

DATA_BLOCK "Btn_STOP"   // DB81
{ S7_Optimized_Access := 'FALSE' }
AUTHOR : Dmitriy_Petrov
VERSION : 0.1
// Кнопка СТОП
// stored: InstanceOfName READ_DISCRET_SIGNAL
"READ_DISCRET_SIGNAL"
BEGIN
   N_module := 8;
   N_chanel := 7;
END_DATA_BLOCK

DATA_BLOCK "Btn_Ventilation"   // DB82
{ S7_Optimized_Access := 'FALSE' }
AUTHOR : Dmitriy_Petrov
VERSION : 0.1
// Кнопка Вентиляция
// stored: InstanceOfName READ_DISCRET_SIGNAL
"READ_DISCRET_SIGNAL"
BEGIN
   N_module := 8;
   N_chanel := 8;
END_DATA_BLOCK

DATA_BLOCK "Btn_Ignition"   // DB83
{ S7_Optimized_Access := 'FALSE' }
AUTHOR : Dmitriy_Petrov
VERSION : 0.1
// Кнопка Розжиг
// stored: InstanceOfName READ_DISCRET_SIGNAL
"READ_DISCRET_SIGNAL"
BEGIN
   N_module := 8;
   N_chanel := 9;
END_DATA_BLOCK

DATA_BLOCK "Btn_Sound"   // DB84
{ S7_Optimized_Access := 'FALSE' }
AUTHOR : Dmitriy_Petrov
VERSION : 0.1
// Кнопка Сброс звука / Проверка звука
// stored: InstanceOfName READ_DISCRET_SIGNAL
"READ_DISCRET_SIGNAL"
BEGIN
   N_module := 8;
   N_chanel := 10;
END_DATA_BLOCK

DATA_BLOCK "ZRW_open"   // DB85
{ S7_Optimized_Access := 'FALSE' }
AUTHOR : Dmitriy_Petrov
VERSION : 0.1
// Регулирующая заслонка питательной воды на котел открыта
// stored: InstanceOfName READ_DISCRET_SIGNAL
"READ_DISCRET_SIGNAL"
BEGIN
   N_module := 8;
   N_chanel := 11;
END_DATA_BLOCK

DATA_BLOCK "ZRW_close"   // DB86
{ S7_Optimized_Access := 'FALSE' }
AUTHOR : Dmitriy_Petrov
VERSION : 0.1
// Регулирующая заслонка питательной воды на котел закрыта
// stored: InstanceOfName READ_DISCRET_SIGNAL
"READ_DISCRET_SIGNAL"
BEGIN
   N_module := 8;
   N_chanel := 12;
END_DATA_BLOCK

DATA_BLOCK "ZRW_middle"   // DB87
{ S7_Optimized_Access := 'FALSE' }
AUTHOR : Dmitriy_Petrov
VERSION : 0.1
// Регулирующая заслонка питательной воды на котел среднее
// stored: InstanceOfName READ_DISCRET_SIGNAL
"READ_DISCRET_SIGNAL"
BEGIN
   N_module := 8;
   N_chanel := 13;
END_DATA_BLOCK

DATA_BLOCK "ZRW_avto"   // DB88
{ S7_Optimized_Access := 'FALSE' }
AUTHOR : Dmitriy_Petrov
VERSION : 0.1
// Регулирующая заслонка питательной воды на котел. БРУ в положении "Авт"
// stored: InstanceOfName READ_DISCRET_SIGNAL
"READ_DISCRET_SIGNAL"
BEGIN
   N_module := 8;
   N_chanel := 14;
END_DATA_BLOCK

DATA_BLOCK "Power_PLC_from_UPS"   // DB89
{ S7_Optimized_Access := 'FALSE' }
AUTHOR : Dmitriy_Petrov
VERSION : 0.1
// Питание контроллера от ИБП
// stored: InstanceOfName READ_DISCRET_SIGNAL
"READ_DISCRET_SIGNAL"
BEGIN
   N_module := 8;
   N_chanel := 15;
END_DATA_BLOCK

DATA_BLOCK "UPS_Low_charge"   // DB90
{ S7_Optimized_Access := 'FALSE' }
AUTHOR : Dmitriy_Petrov
VERSION : 0.1
// Заряд батареи ИБП низкий
// stored: InstanceOfName READ_DISCRET_SIGNAL
"READ_DISCRET_SIGNAL"
BEGIN
   N_module := 8;
   N_chanel := 16;
END_DATA_BLOCK

DATA_BLOCK "ZRG_voltage_ok"   // DB91
{ S7_Optimized_Access := 'FALSE' }
AUTHOR : Dmitriy_Petrov
VERSION : 0.1
// ЗРГ Напряжение в норме
// stored: InstanceOfName READ_DISCRET_SIGNAL
"READ_DISCRET_SIGNAL"
BEGIN
   N_module := 9;
   N_chanel := 1;
END_DATA_BLOCK

DATA_BLOCK "NAV_voltage_ok"   // DB92
{ S7_Optimized_Access := 'FALSE' }
AUTHOR : Dmitriy_Petrov
VERSION : 0.1
// НАВ Напряжение в норме
// stored: InstanceOfName READ_DISCRET_SIGNAL
"READ_DISCRET_SIGNAL"
BEGIN
   N_module := 9;
   N_chanel := 2;
END_DATA_BLOCK

DATA_BLOCK "NAD_voltage_ok"   // DB93
{ S7_Optimized_Access := 'FALSE' }
AUTHOR : Dmitriy_Petrov
VERSION : 0.1
// НАД Напряжение в норме
// stored: InstanceOfName READ_DISCRET_SIGNAL
"READ_DISCRET_SIGNAL"
BEGIN
   N_module := 9;
   N_chanel := 3;
END_DATA_BLOCK

DATA_BLOCK "ZRW_voltage_ok"   // DB94
{ S7_Optimized_Access := 'FALSE' }
AUTHOR : Dmitriy_Petrov
VERSION : 0.1
// ЗРВ Напряжение в норме
// stored: InstanceOfName READ_DISCRET_SIGNAL
"READ_DISCRET_SIGNAL"
BEGIN
   N_module := 9;
   N_chanel := 4;
END_DATA_BLOCK

DATA_BLOCK "SHEU_voltage_ok"   // DB95
{ S7_Optimized_Access := 'FALSE' }
AUTHOR : Dmitriy_Petrov
VERSION : 0.1
// Контроль питания сети ~400В 1ШЭУ
// stored: InstanceOfName READ_DISCRET_SIGNAL
"READ_DISCRET_SIGNAL"
BEGIN
   N_module := 10;
   N_chanel := 12;
END_DATA_BLOCK

DATA_BLOCK "ZDG_no_open"   // DB96
{ S7_Optimized_Access := 'FALSE' }
AUTHOR : Dmitriy_Petrov
VERSION : 0.1
// ЗДГ перед БГ. не открыта
// stored: InstanceOfName READ_DISCRET_SIGNAL
"READ_DISCRET_SIGNAL"
BEGIN
   N_module := 9;
   N_chanel := 6;
END_DATA_BLOCK

DATA_BLOCK "ZDG_no_close"   // DB97
{ S7_Optimized_Access := 'FALSE' }
AUTHOR : Dmitriy_Petrov
VERSION : 0.1
// ЗДГ перед БГ. не закрыта
// stored: InstanceOfName READ_DISCRET_SIGNAL
"READ_DISCRET_SIGNAL"
BEGIN
   N_module := 9;
   N_chanel := 7;
END_DATA_BLOCK

DATA_BLOCK "ZDG_opening"   // DB98
{ S7_Optimized_Access := 'FALSE' }
AUTHOR : Dmitriy_Petrov
VERSION : 0.1
// ЗДГ перед БГ. ход открытие
// stored: InstanceOfName READ_DISCRET_SIGNAL
"READ_DISCRET_SIGNAL"
BEGIN
   N_module := 9;
   N_chanel := 8;
END_DATA_BLOCK

DATA_BLOCK "ZDG_closing"   // DB99
{ S7_Optimized_Access := 'FALSE' }
AUTHOR : Dmitriy_Petrov
VERSION : 0.1
// ЗДГ перед БГ. ход закрытие
// stored: InstanceOfName READ_DISCRET_SIGNAL
"READ_DISCRET_SIGNAL"
BEGIN
   N_module := 9;
   N_chanel := 9;
END_DATA_BLOCK

DATA_BLOCK "ZDG_voltage_ok"   // DB100
{ S7_Optimized_Access := 'FALSE' }
AUTHOR : Dmitriy_Petrov
VERSION : 0.1
// ЗДГ перед БГ. Напряжение в норме
// stored: InstanceOfName READ_DISCRET_SIGNAL
"READ_DISCRET_SIGNAL"
BEGIN
   N_module := 9;
   N_chanel := 10;
END_DATA_BLOCK

DATA_BLOCK "ZDSV_before_boiler_no_open"   // DB101
{ S7_Optimized_Access := 'FALSE' }
AUTHOR : Dmitriy_Petrov
VERSION : 0.1
// ЗДСВ перед котлом. не открыта
// stored: InstanceOfName READ_DISCRET_SIGNAL
"READ_DISCRET_SIGNAL"
BEGIN
   N_module := 9;
   N_chanel := 11;
END_DATA_BLOCK

DATA_BLOCK "ZDSV_before_boiler_no_close"   // DB102
{ S7_Optimized_Access := 'FALSE' }
AUTHOR : Dmitriy_Petrov
VERSION : 0.1
// ЗДСВ перед котлом. не закрыта
// stored: InstanceOfName READ_DISCRET_SIGNAL
"READ_DISCRET_SIGNAL"
BEGIN
   N_module := 9;
   N_chanel := 12;
   Invert := true;
END_DATA_BLOCK

DATA_BLOCK "ZDSV_before_boiler_opening"   // DB103
{ S7_Optimized_Access := 'FALSE' }
AUTHOR : Dmitriy_Petrov
VERSION : 0.1
// ЗДСВ перед котлом. ход открытие
// stored: InstanceOfName READ_DISCRET_SIGNAL
"READ_DISCRET_SIGNAL"
BEGIN
   N_module := 9;
   N_chanel := 13;
END_DATA_BLOCK

DATA_BLOCK "ZDSV_before_boiler_closing"   // DB104
{ S7_Optimized_Access := 'FALSE' }
AUTHOR : Dmitriy_Petrov
VERSION : 0.1
// ЗДСВ перед котлом. ход закрытие
// stored: InstanceOfName READ_DISCRET_SIGNAL
"READ_DISCRET_SIGNAL"
BEGIN
   N_module := 9;
   N_chanel := 14;
END_DATA_BLOCK

DATA_BLOCK "ZDSV_before_boiler_voltage_ok"   // DB105
{ S7_Optimized_Access := 'FALSE' }
AUTHOR : Dmitriy_Petrov
VERSION : 0.1
// ЗДСВ перед котлом. Напряжение в норме
// stored: InstanceOfName READ_DISCRET_SIGNAL
"READ_DISCRET_SIGNAL"
BEGIN
   N_module := 9;
   N_chanel := 15;
END_DATA_BLOCK

DATA_BLOCK "ZDSV_before_boiler_limit_rotational_moment"   // DB106
{ S7_Optimized_Access := 'FALSE' }
AUTHOR : Dmitriy_Petrov
VERSION : 0.1
// ЗДСВ перед котлом. ограничитель крутящего момента
// stored: InstanceOfName READ_DISCRET_SIGNAL
"READ_DISCRET_SIGNAL"
BEGIN
   N_module := 9;
   N_chanel := 16;
END_DATA_BLOCK

DATA_BLOCK "GPZ_no_open"   // DB107
{ S7_Optimized_Access := 'FALSE' }
AUTHOR : Dmitriy_Petrov
VERSION : 0.1
// ГПЗ. не открыта
// stored: InstanceOfName READ_DISCRET_SIGNAL
"READ_DISCRET_SIGNAL"
BEGIN
   N_module := 10;
   N_chanel := 1;
END_DATA_BLOCK

DATA_BLOCK "GPZ_no_close"   // DB108
{ S7_Optimized_Access := 'FALSE' }
AUTHOR : Dmitriy_Petrov
VERSION : 0.1
// ГПЗ. не закрыта
// stored: InstanceOfName READ_DISCRET_SIGNAL
"READ_DISCRET_SIGNAL"
BEGIN
   N_module := 10;
   N_chanel := 2;
END_DATA_BLOCK

DATA_BLOCK "GPZ_opening"   // DB109
{ S7_Optimized_Access := 'FALSE' }
AUTHOR : Dmitriy_Petrov
VERSION : 0.1
// ГПЗ. ход открытие
// stored: InstanceOfName READ_DISCRET_SIGNAL
"READ_DISCRET_SIGNAL"
BEGIN
   N_module := 10;
   N_chanel := 3;
END_DATA_BLOCK

DATA_BLOCK "GPZ_closing"   // DB110
{ S7_Optimized_Access := 'FALSE' }
AUTHOR : Dmitriy_Petrov
VERSION : 0.1
// ГПЗ. ход закрытие
// stored: InstanceOfName READ_DISCRET_SIGNAL
"READ_DISCRET_SIGNAL"
BEGIN
   N_module := 10;
   N_chanel := 4;
END_DATA_BLOCK

DATA_BLOCK "GPZ_voltage_ok"   // DB111
{ S7_Optimized_Access := 'FALSE' }
AUTHOR : Dmitriy_Petrov
VERSION : 0.1
// ГПЗ. Напряжение в норме
// stored: InstanceOfName READ_DISCRET_SIGNAL
"READ_DISCRET_SIGNAL"
BEGIN
   N_module := 10;
   N_chanel := 5;
END_DATA_BLOCK

DATA_BLOCK "GPZ_limit_rotational_moment"   // DB112
{ S7_Optimized_Access := 'FALSE' }
AUTHOR : Dmitriy_Petrov
VERSION : 0.1
// ГПЗ. ограничитель крутящего момента
// stored: InstanceOfName READ_DISCRET_SIGNAL
"READ_DISCRET_SIGNAL"
BEGIN
   N_module := 10;
   N_chanel := 6;
END_DATA_BLOCK

// folder: System blocks/Program resources

DATA_BLOCK "TON_alarm_1_DB"   // DB157
{ S7_Optimized_Access := 'TRUE' }
AUTHOR : Simatic
FAMILY : IEC
NAME : IEC_TMR
VERSION : 1.0
// stored: InstanceOfName IEC_TIMER
"IEC_TIMER"
BEGIN
END_DATA_BLOCK

DATA_BLOCK "TON_alarm_2_DB"   // DB158
{ S7_Optimized_Access := 'TRUE' }
AUTHOR : Simatic
FAMILY : IEC
NAME : IEC_TMR
VERSION : 1.0
// stored: InstanceOfName IEC_TIMER
"IEC_TIMER"
BEGIN
END_DATA_BLOCK

DATA_BLOCK "TON_alarm_3_DB"   // DB159
{ S7_Optimized_Access := 'TRUE' }
AUTHOR : Simatic
FAMILY : IEC
NAME : IEC_TMR
VERSION : 1.0
// stored: InstanceOfName IEC_TIMER
"IEC_TIMER"
BEGIN
END_DATA_BLOCK

DATA_BLOCK "TON_alarm_4_DB"   // DB160
{ S7_Optimized_Access := 'TRUE' }
AUTHOR : Simatic
FAMILY : IEC
NAME : IEC_TMR
VERSION : 1.0
// stored: InstanceOfName IEC_TIMER
"IEC_TIMER"
BEGIN
END_DATA_BLOCK

DATA_BLOCK "TON_alarm_5_DB"   // DB161
{ S7_Optimized_Access := 'TRUE' }
AUTHOR : Simatic
FAMILY : IEC
NAME : IEC_TMR
VERSION : 1.0
// stored: InstanceOfName IEC_TIMER
"IEC_TIMER"
BEGIN
END_DATA_BLOCK

DATA_BLOCK "TON_alarm_6_DB"   // DB162
{ S7_Optimized_Access := 'TRUE' }
AUTHOR : Simatic
FAMILY : IEC
NAME : IEC_TMR
VERSION : 1.0
// stored: InstanceOfName IEC_TIMER
"IEC_TIMER"
BEGIN
END_DATA_BLOCK

DATA_BLOCK "TON_alarm_7_DB"   // DB163
{ S7_Optimized_Access := 'TRUE' }
AUTHOR : Simatic
FAMILY : IEC
NAME : IEC_TMR
VERSION : 1.0
// stored: InstanceOfName IEC_TIMER
"IEC_TIMER"
BEGIN
END_DATA_BLOCK

DATA_BLOCK "TON_alarm_8_DB"   // DB164
{ S7_Optimized_Access := 'TRUE' }
AUTHOR : Simatic
FAMILY : IEC
NAME : IEC_TMR
VERSION : 1.0
// stored: InstanceOfName IEC_TIMER
"IEC_TIMER"
BEGIN
END_DATA_BLOCK

DATA_BLOCK "TON_alarm_9_DB"   // DB165
{ S7_Optimized_Access := 'TRUE' }
AUTHOR : Simatic
FAMILY : IEC
NAME : IEC_TMR
VERSION : 1.0
// stored: InstanceOfName IEC_TIMER
"IEC_TIMER"
BEGIN
END_DATA_BLOCK

DATA_BLOCK "TON_alarm_10_DB"   // DB166
{ S7_Optimized_Access := 'TRUE' }
AUTHOR : Simatic
FAMILY : IEC
NAME : IEC_TMR
VERSION : 1.0
// stored: InstanceOfName IEC_TIMER
"IEC_TIMER"
BEGIN
END_DATA_BLOCK

DATA_BLOCK "TON_alarm_11_DB"   // DB167
{ S7_Optimized_Access := 'TRUE' }
AUTHOR : Simatic
FAMILY : IEC
NAME : IEC_TMR
VERSION : 1.0
// stored: InstanceOfName IEC_TIMER
"IEC_TIMER"
BEGIN
END_DATA_BLOCK

DATA_BLOCK "TON_alarm_12_DB"   // DB168
{ S7_Optimized_Access := 'TRUE' }
AUTHOR : Simatic
FAMILY : IEC
NAME : IEC_TMR
VERSION : 1.0
// stored: InstanceOfName IEC_TIMER
"IEC_TIMER"
BEGIN
END_DATA_BLOCK

DATA_BLOCK "TON_alarm_13_DB"   // DB169
{ S7_Optimized_Access := 'TRUE' }
AUTHOR : Simatic
FAMILY : IEC
NAME : IEC_TMR
VERSION : 1.0
// stored: InstanceOfName IEC_TIMER
"IEC_TIMER"
BEGIN
END_DATA_BLOCK

DATA_BLOCK "TON_alarm_14_DB"   // DB170
{ S7_Optimized_Access := 'TRUE' }
AUTHOR : Simatic
FAMILY : IEC
NAME : IEC_TMR
VERSION : 1.0
// stored: InstanceOfName IEC_TIMER
"IEC_TIMER"
BEGIN
END_DATA_BLOCK

DATA_BLOCK "TON_alarm_15_DB"   // DB171
{ S7_Optimized_Access := 'TRUE' }
AUTHOR : Simatic
FAMILY : IEC
NAME : IEC_TMR
VERSION : 1.0
// stored: InstanceOfName IEC_TIMER
"IEC_TIMER"
BEGIN
END_DATA_BLOCK

DATA_BLOCK "TON_alarm_16_DB"   // DB172
{ S7_Optimized_Access := 'TRUE' }
AUTHOR : Simatic
FAMILY : IEC
NAME : IEC_TMR
VERSION : 1.0
// stored: InstanceOfName IEC_TIMER
"IEC_TIMER"
BEGIN
END_DATA_BLOCK

DATA_BLOCK "TON_alarm_17_DB"   // DB173
{ S7_Optimized_Access := 'TRUE' }
AUTHOR : Simatic
FAMILY : IEC
NAME : IEC_TMR
VERSION : 1.0
// stored: InstanceOfName IEC_TIMER
"IEC_TIMER"
BEGIN
END_DATA_BLOCK

DATA_BLOCK "TON_warning_1_DB"   // DB177
{ S7_Optimized_Access := 'TRUE' }
AUTHOR : Simatic
FAMILY : IEC
NAME : IEC_TMR
VERSION : 1.0
// stored: InstanceOfName IEC_TIMER
"IEC_TIMER"
BEGIN
END_DATA_BLOCK

DATA_BLOCK "TON_warning_2_DB"   // DB178
{ S7_Optimized_Access := 'TRUE' }
AUTHOR : Simatic
FAMILY : IEC
NAME : IEC_TMR
VERSION : 1.0
// stored: InstanceOfName IEC_TIMER
"IEC_TIMER"
BEGIN
END_DATA_BLOCK

DATA_BLOCK "TON_warning_3_DB"   // DB180
{ S7_Optimized_Access := 'TRUE' }
AUTHOR : Simatic
FAMILY : IEC
NAME : IEC_TMR
VERSION : 1.0
// stored: InstanceOfName IEC_TIMER
"IEC_TIMER"
BEGIN
END_DATA_BLOCK

DATA_BLOCK "TON_warning_4_DB"   // DB181
{ S7_Optimized_Access := 'TRUE' }
AUTHOR : Simatic
FAMILY : IEC
NAME : IEC_TMR
VERSION : 1.0
// stored: InstanceOfName IEC_TIMER
"IEC_TIMER"
BEGIN
END_DATA_BLOCK

DATA_BLOCK "TON_warning_5_DB"   // DB182
{ S7_Optimized_Access := 'TRUE' }
AUTHOR : Simatic
FAMILY : IEC
NAME : IEC_TMR
VERSION : 1.0
// stored: InstanceOfName IEC_TIMER
"IEC_TIMER"
BEGIN
END_DATA_BLOCK

DATA_BLOCK "TON_warning_6_DB"   // DB183
{ S7_Optimized_Access := 'TRUE' }
AUTHOR : Simatic
FAMILY : IEC
NAME : IEC_TMR
VERSION : 1.0
// stored: InstanceOfName IEC_TIMER
"IEC_TIMER"
BEGIN
END_DATA_BLOCK

DATA_BLOCK "TON_warning_7_DB"   // DB184
{ S7_Optimized_Access := 'TRUE' }
AUTHOR : Simatic
FAMILY : IEC
NAME : IEC_TMR
VERSION : 1.0
// stored: InstanceOfName IEC_TIMER
"IEC_TIMER"
BEGIN
END_DATA_BLOCK

DATA_BLOCK "TON_warning_8_DB"   // DB185
{ S7_Optimized_Access := 'TRUE' }
AUTHOR : Simatic
FAMILY : IEC
NAME : IEC_TMR
VERSION : 1.0
// stored: InstanceOfName IEC_TIMER
"IEC_TIMER"
BEGIN
END_DATA_BLOCK

DATA_BLOCK "TON_test_sound_DB"   // DB205
{ S7_Optimized_Access := 'TRUE' }
AUTHOR : Simatic
FAMILY : IEC
NAME : IEC_TMR
VERSION : 1.0
// stored: InstanceOfName IEC_TIMER
"IEC_TIMER"
BEGIN
END_DATA_BLOCK

DATA_BLOCK "TON_protection_13_DB"   // DB217
{ S7_Optimized_Access := 'TRUE' }
AUTHOR : Simatic
FAMILY : IEC
NAME : IEC_TMR
VERSION : 1.0
// stored: InstanceOfName IEC_TIMER
"IEC_TIMER"
BEGIN
END_DATA_BLOCK

DATA_BLOCK "TOF_Log_DB"   // DB220
{ S7_Optimized_Access := 'TRUE' }
AUTHOR : Simatic
FAMILY : IEC
NAME : IEC_TMR
VERSION : 1.0
// stored: InstanceOfName IEC_TIMER
"IEC_TIMER"
BEGIN
END_DATA_BLOCK

DATA_BLOCK "TON_close_KZ_DB"   // DB250
{ S7_Optimized_Access := 'TRUE' }
AUTHOR : Simatic
FAMILY : IEC
NAME : IEC_TMR
VERSION : 1.0
// stored: InstanceOfName IEC_TIMER
"IEC_TIMER"
BEGIN
END_DATA_BLOCK

DATA_BLOCK "TON_avto_reset_IVN_DB"   // DB252
{ S7_Optimized_Access := 'TRUE' }
AUTHOR : Simatic
FAMILY : IEC
NAME : IEC_TMR
VERSION : 1.0
// stored: InstanceOfName IEC_TIMER
"IEC_TIMER"
BEGIN
END_DATA_BLOCK

DATA_BLOCK "Timer_IND_1_DB"   // DB260
{ S7_Optimized_Access := 'TRUE' }
AUTHOR : Simatic
FAMILY : IEC
NAME : IEC_TMR
VERSION : 1.0
// stored: InstanceOfName IEC_TIMER
"IEC_TIMER"
BEGIN
END_DATA_BLOCK

DATA_BLOCK "Timer_IND_2_DB"   // DB261
{ S7_Optimized_Access := 'TRUE' }
AUTHOR : Simatic
FAMILY : IEC
NAME : IEC_TMR
VERSION : 1.0
// stored: InstanceOfName IEC_TIMER
"IEC_TIMER"
BEGIN
END_DATA_BLOCK

DATA_BLOCK "Timer_VENTILATION_temp_DB"   // DB262
{ S7_Optimized_Access := 'TRUE' }
AUTHOR : Simatic
FAMILY : IEC
NAME : IEC_TMR
VERSION : 1.0
// stored: InstanceOfName IEC_TIMER
"IEC_TIMER"
BEGIN
END_DATA_BLOCK

DATA_BLOCK "Timer_VENTILATION_DB"   // DB263
{ S7_Optimized_Access := 'TRUE' }
AUTHOR : Simatic
FAMILY : IEC
NAME : IEC_TMR
VERSION : 1.0
// stored: InstanceOfName IEC_TIMER
"IEC_TIMER"
BEGIN
END_DATA_BLOCK

DATA_BLOCK "Timer_PRESS_temp_DB"   // DB264
{ S7_Optimized_Access := 'TRUE' }
AUTHOR : Simatic
FAMILY : IEC
NAME : IEC_TMR
VERSION : 1.0
// stored: InstanceOfName IEC_TIMER
"IEC_TIMER"
BEGIN
END_DATA_BLOCK

DATA_BLOCK "Timer_HEATING_temp_DB"   // DB265
{ S7_Optimized_Access := 'TRUE' }
AUTHOR : Simatic
FAMILY : IEC
NAME : IEC_TMR
VERSION : 1.0
// stored: InstanceOfName IEC_TIMER
"IEC_TIMER"
BEGIN
END_DATA_BLOCK

DATA_BLOCK "Timer_RUN_temp_DB"   // DB266
{ S7_Optimized_Access := 'TRUE' }
AUTHOR : Simatic
FAMILY : IEC
NAME : IEC_LTMR
VERSION : 1.0
// stored: InstanceOfName IEC_LTIMER
"IEC_LTIMER"
BEGIN
END_DATA_BLOCK

DATA_BLOCK "Timer_SHORT_VENTILATION_temp_DB"   // DB267
{ S7_Optimized_Access := 'TRUE' }
AUTHOR : Simatic
FAMILY : IEC
NAME : IEC_TMR
VERSION : 1.0
// stored: InstanceOfName IEC_TIMER
"IEC_TIMER"
BEGIN
END_DATA_BLOCK

DATA_BLOCK "Timer_IGNITION_temp_DB"   // DB268
{ S7_Optimized_Access := 'TRUE' }
AUTHOR : Simatic
FAMILY : IEC
NAME : IEC_TMR
VERSION : 1.0
// stored: InstanceOfName IEC_TIMER
"IEC_TIMER"
BEGIN
END_DATA_BLOCK

DATA_BLOCK "Timer_IGNITION_control_flame_DB"   // DB269
{ S7_Optimized_Access := 'TRUE' }
AUTHOR : Simatic
FAMILY : IEC
NAME : IEC_TMR
VERSION : 1.0
// stored: InstanceOfName IEC_TIMER
"IEC_TIMER"
BEGIN
END_DATA_BLOCK

DATA_BLOCK "Timer_MIN_POWER_temp_DB"   // DB270
{ S7_Optimized_Access := 'TRUE' }
AUTHOR : Simatic
FAMILY : IEC
NAME : IEC_TMR
VERSION : 1.0
// stored: InstanceOfName IEC_TIMER
"IEC_TIMER"
BEGIN
END_DATA_BLOCK

DATA_BLOCK "Timer_MIN_POWER_1_DB"   // DB271
{ S7_Optimized_Access := 'TRUE' }
AUTHOR : Simatic
FAMILY : IEC
NAME : IEC_TMR
VERSION : 1.0
// stored: InstanceOfName IEC_TIMER
"IEC_TIMER"
BEGIN
END_DATA_BLOCK

DATA_BLOCK "Timer_MIN_POWER_2_DB"   // DB272
{ S7_Optimized_Access := 'TRUE' }
AUTHOR : Simatic
FAMILY : IEC
NAME : IEC_TMR
VERSION : 1.0
// stored: InstanceOfName IEC_TIMER
"IEC_TIMER"
BEGIN
END_DATA_BLOCK

DATA_BLOCK "Timer_EMERGENCY_STOP_temp_DB"   // DB273
{ S7_Optimized_Access := 'TRUE' }
AUTHOR : Simatic
FAMILY : IEC
NAME : IEC_TMR
VERSION : 1.0
// stored: InstanceOfName IEC_TIMER
"IEC_TIMER"
BEGIN
END_DATA_BLOCK

DATA_BLOCK "Timer_ALARM_STOP_temp_DB"   // DB274
{ S7_Optimized_Access := 'TRUE' }
AUTHOR : Simatic
FAMILY : IEC
NAME : IEC_TMR
VERSION : 1.0
// stored: InstanceOfName IEC_TIMER
"IEC_TIMER"
BEGIN
END_DATA_BLOCK

DATA_BLOCK "Timer_PLAN_STOP_temp_DB"   // DB275
{ S7_Optimized_Access := 'TRUE' }
AUTHOR : Simatic
FAMILY : IEC
NAME : IEC_TMR
VERSION : 1.0
// stored: InstanceOfName IEC_TIMER
"IEC_TIMER"
BEGIN
END_DATA_BLOCK

DATA_BLOCK "Timer_STOP_PRESS_temp_DB"   // DB276
{ S7_Optimized_Access := 'TRUE' }
AUTHOR : Simatic
FAMILY : IEC
NAME : IEC_TMR
VERSION : 1.0
// stored: InstanceOfName IEC_TIMER
"IEC_TIMER"
BEGIN
END_DATA_BLOCK

DATA_BLOCK "Timer_STOP_MIN_POWER_1_DB"   // DB278
{ S7_Optimized_Access := 'TRUE' }
AUTHOR : Simatic
FAMILY : IEC
NAME : IEC_TMR
VERSION : 1.0
// stored: InstanceOfName IEC_TIMER
"IEC_TIMER"
BEGIN
END_DATA_BLOCK

DATA_BLOCK "Timer_STOP_MIN_POWER_2_DB"   // DB279
{ S7_Optimized_Access := 'TRUE' }
AUTHOR : Simatic
FAMILY : IEC
NAME : IEC_TMR
VERSION : 1.0
// stored: InstanceOfName IEC_TIMER
"IEC_TIMER"
BEGIN
END_DATA_BLOCK

DATA_BLOCK "TON_warning_9_DB"   // DB280
{ S7_Optimized_Access := 'TRUE' }
AUTHOR : Simatic
FAMILY : IEC
NAME : IEC_TMR
VERSION : 1.0
// stored: InstanceOfName IEC_TIMER
"IEC_TIMER"
BEGIN
END_DATA_BLOCK

DATA_BLOCK "TON_warning_10"   // DB281
{ S7_Optimized_Access := 'TRUE' }
AUTHOR : Simatic
FAMILY : IEC
NAME : IEC_TMR
VERSION : 1.0
// stored: InstanceOfName IEC_TIMER
"IEC_TIMER"
BEGIN
END_DATA_BLOCK

DATA_BLOCK "Timer_сlose_GPZ_DB"   // DB285
{ S7_Optimized_Access := 'TRUE' }
AUTHOR : Simatic
FAMILY : IEC
NAME : IEC_TMR
VERSION : 1.0
// stored: InstanceOfName IEC_TIMER
"IEC_TIMER"
BEGIN
END_DATA_BLOCK

// folder: (top level)

FUNCTION_BLOCK "READ_DISCRET_SIGNAL"   // FB1, SCL
{ S7_Optimized_Access := 'FALSE' }
AUTHOR : Dmitriy_Petrov
VERSION : 0.1
// Функциональный блок чтения дискретного параметра
   VAR_INPUT
      Invert : Bool;   // Инвертирование сигнала
      Enable : Bool := TRUE;   // Разрешение использования параметра
   END_VAR
   VAR_OUTPUT
      Value : Bool;   // Значение сигнала
   END_VAR
   VAR_IN_OUT
      N_module : USInt;   // № модуля (начиная с 1)
      N_chanel : USInt;   // № канала (начиная с 1)
   END_VAR
BEGIN
   #Value:="read_discret"(Invert :=#Invert, N_module :=#N_module, N_chanel :=#N_chanel);
END_FUNCTION_BLOCK

FUNCTION_BLOCK "PID_analog"   // FB2, SCL
{ S7_Optimized_Access := 'FALSE' }
VERSION : 0.1
   VAR_INPUT
      AUTO : Bool;   // Mode (0-manual, 1-automatic)
      DIR : Bool;   // Direction (1-positive,0-negative)
      PV : Real;   // Process variable
      SP : Real;   // Setpoint
      DB : Real;   // Deadband
      KP : Real;   // Proportional constant
      TI : UDInt;   // Integral time constant (ms)
      TD : UDInt;   // Derivative time constant (ms)
      CYCLE : UDInt;   // Cycle time (ms)
      OUT_MIN : Real;   // Output min limit (automatic mode)
      OUT_MAX : Real := 100.0;   // Output max limit (automatic mode)
      OUT_MAN : Real;   // Output (manual mode)
      Hold : Bool;   // (1-заморозка, 0-выполнение)
   END_VAR
   VAR_IN_OUT
      OUT : Real;   // Output control
   END_VAR
   VAR
      Err : Real;   // Ошибка рассогласования (t)
      Err_T : Real;   // Предыдущее значение ошибки рассогласования (t-1)
      Out_T : Real;   // Предыдущее значение выхода (t-1)
      Er : Real;   // Ошибка рассогласования (t)
      Er_T : Real;   // Предыдущее значение ошибки рассогласования (t-1)
      Integral : Real;   // Интегральная составляющая (t)
      Integral_T : Real;   // Интегральная составляющая (t-1)
      Integral_D : Real;   // Интегральное изменение
      Pulse : Bool;   // Триггер импульса расчета
      TE : UDInt;
      Reset : Bool;
      KPd : Real;
      A_N : Real := 8.0;
      A_Xf_1 : Real;
      A_Xf_2 : Real;
      Diff : Real;
   END_VAR
BEGIN
   (*Реальное время*)
   IF NOT #Reset THEN
       #TE := 0;
       #Reset := TRUE;
   ELSE
       #TE := #TE + "RT_INFO_DB".Cycle;
   END_IF;
   IF #TE >= #CYCLE AND #CYCLE <> 0 THEN
       #Pulse := TRUE;
   ELSE
       #Pulse := FALSE;
   END_IF;

   (*ПИД регулятор*)
   IF #Pulse THEN
       #Err := #SP - #PV;
       #Er := #Err;
       IF NOT #Hold THEN
           IF NOT #DIR THEN
               #KPd := INT_TO_REAL(0) - #KP;
           ELSE
               #KPd := #KP;
           END_IF;
           IF #AUTO THEN
               IF ABS(#Er) < #DB / INT_TO_REAL(10) THEN
                   #Err := INT_TO_REAL(0);
                   #Err_T := INT_TO_REAL(0);
               END_IF;
               IF ABS(#Er) > #DB / INT_TO_REAL(2) THEN
                   #Err := #Er;
               END_IF;
               IF ABS(#Er) <= #DB / INT_TO_REAL(2) AND ABS(#Er) >= #DB / INT_TO_REAL(10) THEN
                   IF #Err_T = INT_TO_REAL(0) THEN
                       #Err := INT_TO_REAL(0);
                       #Err_T := INT_TO_REAL(0);
                   ELSE
                       #Err := #Er;
                   END_IF;
               END_IF;
               IF #TI <= 0 THEN
                   #Integral_T := INT_TO_REAL(0);
                   #Integral_D := INT_TO_REAL(0);
                   #Integral := INT_TO_REAL(0);
               ELSE
                   #Integral_D := #KPd * ((#Err * UDINT_TO_REAL(#TE)) / UDINT_TO_REAL(#TI));
                   #Integral := #Integral_T + #Integral_D;
               END_IF;
               IF #TD > 0 THEN
                   (*Фильтр 1-го порядка (Апериодическое звено)*)
                   #A_Xf_1 := #A_Xf_1 + (#Err - #A_Xf_1) * UDINT_TO_REAL(#TE) / (UDINT_TO_REAL(#TD) / #A_N + UDINT_TO_REAL(#TE));
                   (*Фильтр 2-го порядка (Апериодическое звено)*)
                   #A_Xf_2 := #A_Xf_2 + (#Err - #A_Xf_1 - #A_Xf_2) * UDINT_TO_REAL(#TE) / (UDINT_TO_REAL(#TD) / #A_N + UDINT_TO_REAL(#TE));
                   #Diff := #KPd * #A_N * #A_Xf_2;
               ELSE
                   #A_Xf_1 := #Err;
                   #Diff := INT_TO_REAL(0);
               END_IF;
               #OUT := #KPd * #Err + #Integral + #Diff;
               IF #OUT < #OUT_MIN THEN
                   IF #Integral_D < INT_TO_REAL(0) THEN
                       #Integral_D := INT_TO_REAL(0);
                   END_IF;
               END_IF;
               IF #OUT > #OUT_MAX THEN
                   IF #Integral_D > INT_TO_REAL(0) THEN
                       #Integral_D := INT_TO_REAL(0);
                   END_IF;
               END_IF;
               #Integral := #Integral_T + #Integral_D;
               #OUT := #KPd * #Err + #Integral + #Diff;
               IF #OUT < #OUT_MIN THEN
                   #OUT := #OUT_MIN;
               END_IF;
               IF #OUT > #OUT_MAX THEN
                   #OUT := #OUT_MAX;
               END_IF;
           ELSE
               #OUT := #OUT_MAN;
               IF #OUT < #OUT_MIN THEN
                   #OUT := #OUT_MIN;
               END_IF;
               IF #OUT > #OUT_MAX THEN
                   #OUT := #OUT_MAX;
               END_IF;
               #Integral := #OUT - #KPd * #Err;
               #A_Xf_1 := INT_TO_REAL(0);
               #A_Xf_2 := INT_TO_REAL(0);
           END_IF;
           (*Проверка ошибок*)
           ENO := TRUE;    //ENO := NOT P_ER;
       ELSE
           #Err := INT_TO_REAL(0);
           #Err_T := INT_TO_REAL(0);
           #OUT := #OUT_MIN;
           #Integral := INT_TO_REAL(0);
       END_IF;
       #Err_T := #Err;
       #Er_T := #Er;
       #Out_T := #OUT;
       #Integral_T := #Integral;
       #TE := 0;
   END_IF;
END_FUNCTION_BLOCK

FUNCTION_BLOCK "TIME_converter"   // FB3, SCL
{ S7_Optimized_Access := 'FALSE' }
VERSION : 0.1
   VAR_INPUT
      IN : Time;   // входная переменная тип Time
   END_VAR
   VAR_OUTPUT
      Hour : Int;   // Часы
      Minute : Int;   // Минуты
      Second : Int;   // Секунды
   END_VAR
   VAR_TEMP
      in_dint_ms : DInt;
      in_dint_s : DInt;
      in_dint_m : DInt;
      in_dint_h : DInt;
   END_VAR
BEGIN
   #in_dint_ms := T_CONV(#IN);
   #in_dint_s := #in_dint_ms / 1000;
   #in_dint_m := #in_dint_s / 60;
   #in_dint_h := #in_dint_m / 60;

   #Second := DINT_TO_INT((#in_dint_s) MOD (60));
   #Minute := DINT_TO_INT((#in_dint_m) MOD (60));
   #Hour := DINT_TO_INT(#in_dint_h);
END_FUNCTION_BLOCK

FUNCTION_BLOCK "LTIME_converter"   // FB4, SCL
{ S7_Optimized_Access := 'FALSE' }
VERSION : 0.1
   VAR_INPUT
      IN : LTime;   // входная переменная тип LTime
   END_VAR
   VAR_OUTPUT
      Day : DInt;   // Дни
      Hour : Int;   // Часы
      Minute : Int;   // Минуты
      Second : Int;   // Секунды
      mSecond : Int;   // Миллисекунды
      uSecond : Int;   // Микросекунды
      nSecond : Int;   // Наносекунды
   END_VAR
   VAR_TEMP
      temp_ns : LInt;
      temp_us : LInt;
      temp_ms : LInt;
      temp_s : LInt;
      temp_m : LInt;
      temp_h : LInt;
      temp_d : LInt;
   END_VAR
BEGIN
   #temp_ns := T_CONV(#IN);
   #temp_us := #temp_ns / 1000;
   #temp_ms := #temp_us / 1000;
   #temp_s := #temp_ms / 1000;
   #temp_m := #temp_s / 60;
   #temp_h := #temp_m / 60;
   #temp_d := #temp_h / 24;

   #nSecond := LINT_TO_INT((#temp_ns) MOD (1000));
   #uSecond := LINT_TO_INT((#temp_us) MOD (1000));
   #mSecond := LINT_TO_INT((#temp_ms) MOD (1000));
   #Second := LINT_TO_INT((#temp_s) MOD (60));
   #Minute := LINT_TO_INT((#temp_m) MOD (60));
   #Hour := LINT_TO_INT((#temp_h) MOD (24));
   #Day := LINT_TO_DINT(#temp_d);
END_FUNCTION_BLOCK

FUNCTION_BLOCK "PID_impulse"   // FB5, SCL
{ S7_Optimized_Access := 'FALSE' }
VERSION : 0.1
   VAR_INPUT
      DIR : Bool;   // Направление регулирования (1-позитивное,0-негативное)
      PV : Real;   // Величина параметра
      SP : Real;   // Величина уставки
      DB : Real;   // Зона нечувствительности
      KP : Real;   // ПИД Пропорциональный коэффициент
      TI : UDInt;   // ПИД Постоянная времени интегрирования (мс)
      TD : UDInt;   // ПИД Постоянная времени дифференцирования (мс)
      CYCLE : UDInt;   // Время цикла регулятора (мс)
      FMT : UDInt;   // Время хода исполнительного механизма (мс)
      DT_MIN : UDInt;   // Величина минимальной длительности импульса (мс)
      AUTO : Bool;   // Режим работы (0-ДИСТ, 1- АВТ)
      MORE : Bool;   // Дистанционное управление. Кнопка "Больше"
      LESS : Bool;   // Дистанционное управление. Кнопка "Меньше"
      Hold : Bool;   // (1-заморозка, 0-выполнение)
      GAP : DInt;   // Люфт
   END_VAR
   VAR_IN_OUT
      PLUS : Bool;   // Управление "Больше"
      MINUS : Bool;   // Управление "Меньше"
   END_VAR
   VAR
      BDP : Real;
      dD : Real;   // Приращение дифференциальной составляющей
      dD_max : Real;
      dI : Real;   // Приращение интегральной составляющей
      dP : Real;   // Приращение пропорциональной составляющей
      dP_1 : Real;
      dt10 : DInt;
      dt2_T : DInt;
      dt3 : DInt;
      dt3_T : DInt;
      dt4 : DInt;
      dt7 : DInt;
      dt8 : DInt;
      dt_imp_T : DInt;
      Err : Real;   // Ошибка рассогласования (t)
      Err_1 : Real;
      Err_1_T : Real;
      Ik : DInt;
      Int_reset : Bool;
      KPd : Real;
      L5 : Bool;
      L5_T : Bool;
      out : Bool;
      Pulse : Bool;   // Триггер импульса расчета
      Reset : Bool;
      TE : UDInt;   // Время цикла регулятора
      dP_T : Real;
      dI_T : Real;
      D_T : Real;
      A_N : Real := 8.0;
      A_Xf_1 : Real;
      A_Xf_2 : Real;
      D : Real;   // Приращение дифференциальной составляющей
      dD_1 : Real;
      dU : Real;   // Приращение управляющего воздействия
      dt1 : DInt;   // Длительность импульса
      dt6 : DInt;
      dt_imp : DInt;
      PLUS_T : Bool;
      MINUS_T : Bool;
      PAUSE : DInt;   // Время цикла регулятора
      L11 : Bool;
      L12 : Bool;
      Direct : Bool;   // Направление движения механизма (0-больше, 1-меньше)
   END_VAR
BEGIN
   (*Реальное время*)
   IF NOT #Reset THEN
       #TE := 0;
       #Reset := TRUE;
   ELSE
       #TE := #TE + "RT_INFO_DB".Cycle;
   END_IF;
   IF #TE >= #CYCLE AND #CYCLE <> 0 THEN
       #Pulse := TRUE;
   ELSE
       #Pulse := FALSE;
   END_IF;

   (*ПИД регулятор*)
   IF #Pulse THEN
       IF NOT #Hold THEN
           IF #AUTO THEN
               IF NOT #DIR THEN
                   #KPd := INT_TO_REAL(0) - #KP;
               ELSE
                   #KPd := #KP;
               END_IF;
               #Err := #SP - #PV;
               (*Зона нечувствительности*)
               IF ABS(#Err) < #DB / INT_TO_REAL(10) THEN
                   #Err_1 := INT_TO_REAL(0);
                   #Err_1_T := INT_TO_REAL(0);
               END_IF;
               IF ABS(#Err) > #DB / INT_TO_REAL(2) THEN
                   #Err_1 := #Err;
               END_IF;
               IF ABS(#Err) <= #DB / INT_TO_REAL(2) AND ABS(#Err) >= #DB / INT_TO_REAL(10) THEN
                   IF #Err_1_T = INT_TO_REAL(0) THEN
                       #Err_1 := INT_TO_REAL(0);
                       #Err_1_T := INT_TO_REAL(0);
                   ELSE
                       #Err_1 := #Err;
                   END_IF;
               END_IF;
               (*Д*)
               #dP := #KPd * (#Err_1 - #Err_1_T);
               (*Фильтрующий усилитель*)
               IF #TI > 0 THEN
                   #dI := #KPd * (UDINT_TO_REAL(#CYCLE) / UDINT_TO_REAL(#TI)) * ((#Err_1 + #Err_1_T) / INT_TO_REAL(2));
               ELSE
                   #dI := INT_TO_REAL(0);
               END_IF;
               (*ДД*)
               IF #TD > 0 THEN
                   (*Фильтр 1-го порядка (Апериодическое звено)*)
                   #A_Xf_1 := #A_Xf_1 + (#Err_1 - #A_Xf_1) * UDINT_TO_REAL(#CYCLE) / (UDINT_TO_REAL(#TD) / #A_N + UDINT_TO_REAL(#CYCLE));
                   (*Фильтр 2-го порядка (Апериодическое звено)*)
                   #A_Xf_2 := #A_Xf_2 + (#Err_1 - #A_Xf_1 - #A_Xf_2) * UDINT_TO_REAL(#CYCLE) / (UDINT_TO_REAL(#TD) / #A_N + UDINT_TO_REAL(#CYCLE));
                   #D := #KPd * #A_N * #A_Xf_2;
               ELSE
                   #A_Xf_1 := #Err_1;
                   #D := INT_TO_REAL(0);
               END_IF;
               #dD := #D - #D_T;
               (*Блокировка приращения пропорциональной составляющей*)
               #BDP := #KPd * #Err_1;
               IF #dP > INT_TO_REAL(0) AND #BDP < INT_TO_REAL(-100) THEN
                   #dP_1 := INT_TO_REAL(0);
               END_IF;
               IF #dP < INT_TO_REAL(0) AND #BDP > INT_TO_REAL(-100) THEN
                   #dP_1 := INT_TO_REAL(0);
               END_IF;
               IF ABS(#BDP) <= INT_TO_REAL(100) THEN
                   #dP_1 := #dP;
               END_IF;
               (*Ограничение приращений дифференциальной составляющей*)
               IF ABS(#dP_T + #dI_T) < INT_TO_REAL(100) THEN
                   #dD_max := INT_TO_REAL(100) - ABS(#dP_T + #dI_T);
               ELSE
                   #dD_max := INT_TO_REAL(0);
               END_IF;
               IF ABS(#dD) <= #dD_max THEN
                   #dD_1 := #dD;
               END_IF;
               IF #dD > #dD_max THEN
                   #dD_1 := #dD_max;
               END_IF;
               IF #dD < INT_TO_REAL(0) - #dD_max THEN
                   #dD_1 := INT_TO_REAL(0) - #dD_max;
               END_IF;
               (*Формирование ПИД закона*)
               #dU := #dP_1 + #dI + #dD_1;
               (*Ограничение амплитуды*)
               IF #dU < INT_TO_REAL(-100) THEN
                   #dU := INT_TO_REAL(-100);
               END_IF;
               IF #dU > INT_TO_REAL(100) THEN
                   #dU := INT_TO_REAL(100);
               END_IF;
               (*Расчет длительности импульса*)
               #dt1 := REAL_TO_DINT((UDINT_TO_REAL(#FMT) / INT_TO_REAL(100)) * #dU);
               (*Коррекция малых длительностей импульсов*)
               IF ABS(#dt1) < UDINT_TO_DINT(#DT_MIN) THEN
                   #dt3 := #dt1;
               ELSE
                   #dt3 := 0;
               END_IF;
               IF #dt2_T > UDINT_TO_DINT(#DT_MIN) AND ABS(#dt1) < UDINT_TO_DINT(#DT_MIN) THEN
                   #Int_reset := TRUE;
               ELSE
                   #Int_reset := FALSE;
               END_IF;
               #Ik := #Ik + #dt3;
               IF #Int_reset OR #L5_T THEN
                   #Ik := 0;
               END_IF;
               #dt4 := #dt1 + #Ik;
               IF ABS(#dt4) >= UDINT_TO_DINT(#DT_MIN) THEN
                   #L5 := TRUE;
               ELSE
                   #L5 := FALSE;
               END_IF;
               IF NOT #L5 THEN
                   #dt6 := #dt1;
               ELSE
                   #dt6 := #dt4;
               END_IF;
               (*Коррекция больших длительностей импульсов*)
               IF #dt_imp_T >= 0 THEN
                   #dt8 := UDINT_TO_DINT(#CYCLE) - #dt_imp_T;
               ELSE
                   #dt8 := - UDINT_TO_DINT(#CYCLE) - #dt_imp_T;
               END_IF;
               IF ABS(#dt8) > UDINT_TO_DINT(#CYCLE) THEN
                   #dt10 := #dt8;
               ELSE
                   #dt10 := 0;
               END_IF;
               #dt7 := #dt6 - #dt10;
               (*огр амп*)
               IF ABS(#dt7) <= UDINT_TO_DINT(#FMT) THEN
                   #dt_imp := #dt7;
               END_IF;
               IF #dt7 > UDINT_TO_DINT(#FMT) THEN
                   #dt_imp := UDINT_TO_DINT(#FMT);
               END_IF;
               IF #dt7 < - UDINT_TO_DINT(#FMT) THEN
                   #dt_imp := - UDINT_TO_DINT(#FMT);
               END_IF;
   (*Проверка ошибок*)
               ENO := TRUE;    //ENO := NOT P_ER;
           END_IF;
       ELSE
           #Err := INT_TO_REAL(0);
       END_IF;
       #Err_1_T := #Err_1;
       #dt2_T := ABS(#dt1);
       #dt3_T := #dt3;
       #dt_imp_T := #dt_imp;
       #L5_T := #L5;
       #dP_T := #dP;
       #dI_T := #dI;
       #D_T := #D;
       #TE := 0;
   END_IF;

   (* //компенсация люфта
   IF NOT #Direct AND #dt_imp < 0 THEN
       #dt_imp := #dt_imp - #GAP;
   END_IF;
   IF #Direct AND #dt_imp > 0 THEN
       #dt_imp := #dt_imp + #GAP;
   END_IF; *)

   (*Формирование ШИМ выхода*)
   IF #AUTO THEN
       IF UDINT_TO_DINT(#TE) >= ABS(#dt_imp) THEN
           #out := FALSE;
           #PLUS := false;
           #MINUS := false;
       ELSE
           #out := TRUE;
       END_IF;
       IF ABS(#dt_imp) >= UDINT_TO_DINT(#DT_MIN) THEN
           IF #dt_imp > 0 THEN
               IF #out THEN
                   #PLUS := true;
               ELSE
                   #PLUS := false;
               END_IF;
               #MINUS := false;
           ELSE
               IF #out THEN
                   #MINUS := true;
               ELSE
                   #MINUS := false;
               END_IF;
               #PLUS := false;
           END_IF;
   (*    ELSE
           #PLUS := false;
           #MINUS := false; *)
       END_IF;
   ELSE
       #PLUS := #MORE;
       #MINUS := #LESS;
   END_IF;
   (*Защита от частых коммутаций*)
   IF ((#PLUS_T AND NOT #PLUS) OR (#MINUS_T AND NOT #MINUS)) THEN
       #L11 := true;
   END_IF;
   IF #L11 THEN
       #PAUSE := UDINT_TO_DINT(#DT_MIN * INT_TO_UDINT(3));
       #L12 := true;
       #L11 := false;
   END_IF;
   IF #L12 THEN
       IF #PAUSE <= INT_TO_DINT(0) THEN
           #L12 := false;
           #PAUSE := INT_TO_DINT(0);
       ELSE
           #PAUSE := #PAUSE - UDINT_TO_DINT("RT_INFO_DB".Cycle); // / INT_TO_UDINT(10));
       END_IF;
   END_IF;
   IF #L12 AND #AUTO THEN
       #PLUS := false;
       #MINUS := false;
   END_IF;

   #PLUS_T := #PLUS;
   #MINUS_T := #MINUS;

   IF #PLUS THEN
       #Direct := FALSE;
   END_IF;
   IF #MINUS THEN
       #Direct := TRUE;
   END_IF;
END_FUNCTION_BLOCK

FUNCTION_BLOCK "READ_ANALOG_SENSOR"   // FB6, SCL
{ S7_Optimized_Access := 'FALSE' }
AUTHOR : Dmitriy_Petrov
VERSION : 0.1
// Функциональный блок чтения аналогового сигнала
   VAR_INPUT
      LL_sensor_new : Real;   // Нижний предел датчика в физической величине новый
      HL_sensor_new : Real := 100.0;   // Верхний предел датчика в физической величине новый
      LL_ADC_new : Int;   // Нижний предел AЦП новый
      HL_ADC_new : Int := 27648;   // Верхний предел АЦП новый
      Enable_change_limit_online : Bool;   // Разрешение изменять пределы датчика без подтверждения
      Enable : Bool := TRUE;   // Разрешение использования параметра
   END_VAR
   VAR_OUTPUT
      Value : Real;   // Текущее значение в физической величине
      Current : Real;   // Текущее значение тока
      Error_sensor : Bool;   // Неисправность датчика
   END_VAR
   VAR_IN_OUT
      N_module : USInt;   // № модуля (начиная с 1)
      N_chanel : USInt;   // № канала (начиная с 1)
      ADC : Int;   // Текущий код АЦП
      Apply_new_limit : Bool;   // Применить новые пределы датчика
   END_VAR
   VAR
      LL_sensor : Real;   // Нижний предел датчика в физической величине
      HL_sensor : Real := 100.0;   // Верхний предел датчика в физической величине
      LL_ADC : Int;   // Нижний предел АЦП
      HL_ADC : Int := 27648;   // Верхний предел АЦП
   END_VAR
BEGIN
   #Value := "read_4_20"(LL_sensor := #LL_sensor, HL_sensor := #HL_sensor, LL_ADC := #LL_ADC, HL_ADC := #HL_ADC, Current => #Current, error_sensor => #Error_sensor, N_module := #N_module, N_chanel := #N_chanel, ADC := #ADC);

   //применение изменений значений точек для пересчета сигнала
   IF #Enable_change_limit_online THEN
       #LL_sensor := #LL_sensor_new;
       #HL_sensor := #HL_sensor_new;
       #LL_ADC := #LL_ADC_new;
       #HL_ADC := #HL_ADC_new;
       #Apply_new_limit := false;
   ELSE
       IF #Apply_new_limit THEN
           #LL_sensor := #LL_sensor_new;
           #HL_sensor := #HL_sensor_new;
           #LL_ADC := #LL_ADC_new;
           #HL_ADC := #HL_ADC_new;
           #Apply_new_limit := false;
       END_IF;
   END_IF;
END_FUNCTION_BLOCK

FUNCTION_BLOCK "WRITE_ANALOG_SIGNAL"   // FB7, SCL
{ S7_Optimized_Access := 'FALSE' }
AUTHOR : Dmitriy_Petrov
VERSION : 0.1
// Функциональный блок записи аналогового сигнала
   VAR_INPUT
      Value : Real;   // Значение в физической величине
      LL_control_signal_new : Real;   // Нижний предел управляющего воздействия в физической величине новый
      HL_control_signal_new : Real := 100.0;   // Верхний предел управляющего воздействия в физической величине новый
      Enable : Bool := TRUE;   // Разрешение использования параметра
      Enable_change_limit_online : Bool;   // Разрешение изменять пределы датчика без подтверждения
   END_VAR
   VAR_IN_OUT
      N_module : USInt;   // № модуля (начиная с 1)
      N_chanel : USInt;   // № канала (начиная с 1)
      ADC : Int;   // Текущий код АЦП
      Apply_new_limit : Bool;   // Применить новые пределы датчика
   END_VAR
   VAR
      LL_control_signal : Real;   // Нижний предел управляющего воздействия в физической величине
      HL_control_signal : Real := 100.0;   // Верхний предел управляющего воздействия в физической величине
      Current : Real;   // Текущее значение тока
   END_VAR
BEGIN
   "write_4_20"(Value:=#Value,
                LL_control_signal:=#LL_control_signal,
                HL_control_signal:=#HL_control_signal,
                N_module:=#N_module,
                N_chanel:=#N_chanel,
                ADC:=#ADC);

   //применение изменений значений точек для пересчета сигнала
   IF #Enable_change_limit_online THEN
       #LL_control_signal := #LL_control_signal_new;
       #HL_control_signal := #HL_control_signal_new;
       #Apply_new_limit := false;
   ELSE
       IF #Apply_new_limit THEN
           #LL_control_signal := #LL_control_signal_new;
           #HL_control_signal := #HL_control_signal_new;
           #Apply_new_limit := false;
       END_IF;
   END_IF;

   (*вычисление физического значения тока*)
   #Current := (((20 - 4) / (#HL_control_signal - #LL_control_signal)) * #Value) + 4;
END_FUNCTION_BLOCK

FUNCTION_BLOCK "WRITE_DISCRET_SIGNAL"   // FB8, SCL
TITLE = Запись дискретного сигнала
{ S7_Optimized_Access := 'FALSE' }
AUTHOR : Dmitriy_Petrov
VERSION : 0.1
// Функциональный блок записи дискретного параметра
   VAR_INPUT
      Value : Bool;   // Значение сигнала
      Invert : Bool;   // Инвертирование сигнала
      Enable : Bool := TRUE;   // Разрешение использования параметра
   END_VAR
   VAR_IN_OUT
      N_module : USInt;   // № модуля (начиная с 1)
      N_chanel : USInt;   // № канала (начиная с 1)
   END_VAR
BEGIN
   "write_discret"(Value:=#Value,
                   Invert:=#Invert,
                   N_module:=#N_module,
                   N_chanel:=#N_chanel);
END_FUNCTION_BLOCK

FUNCTION_BLOCK "GAS_METER"   // FB9, SCL
{ S7_Optimized_Access := 'FALSE' }
AUTHOR : Петров
VERSION : 0.1
// Счетчик газа с импульсным выходом
   VAR_INPUT
      scale_unit : Real := 100.0;   // Цена одного импульса (литр)
      Time_min_consumption : Time := T#10m;   // Время определения минимального расхода
      consumption_max_value : Real := 100000.0;   // Максимальное показание накопленного расхода [м3]
      Enable : Bool := TRUE;   // Разрешение использования параметра
   END_VAR
   VAR_OUTPUT
      moment_consumption : Real;   // Мгновенный расход (м3/ч)
      dayly_consumption_average : Real;   // Среднесуточное потребление [м3]
   END_VAR
   VAR_IN_OUT
      impulse : Bool;   // Импульсный вход
      impulse_N_module : USInt;   // Импульсный вход № модуля (начиная с 1)
      impulse_N_chanel : USInt;   // Импульсный вход № канала (начиная с 1)
      accumulated_consumption : Real;   // Накопленный расход (м3)
      apply_correct_consumption : Bool;   // Применить скорректированный расход
      correct_consumption : Real;   // Корректировка расхода (м3)
   END_VAR
   VAR
      front_impulse : Bool;   // Фронт импульсного входа
      Moment_consumption_Timer_IN : Bool;   // Таймер вычисления мгновенного расхода. Пуск
      Moment_consumption_Timer_Q : Bool;   // Таймер вычисления мгновенного расхода. Выход
      Moment_consumption_Timer_ET : Time;   // Таймер вычисления мгновенного расхода. Текущее значение
      Time_moment_consumption : Time;   // Время для вычисления мгновенного расхода
      Arhive_consumption : Array[0..3599] of Real;   // Архив 12 минутных расходов
      Arhive_Timer_IN : Bool;   // Таймер архивирования расхода. Пуск
      Arhive_Timer_Q : Bool;   // Таймер архивирования расхода. Выход
      accumulated_consumption_T : Real;   // Накопленный расход в предыдущий момент времени (м3)
      Current_arhive_cunsumption : Real;   // Расход за текущий архивный период [м3]
      Indicator_correct_consumption : Bool;   // Индикатор корректировки показагий расхода
      difference_correct_consumption : Real;   // Изменеие скорректированного расхода (м3)
      marker_arhive : Int;   // Указатель архива
      Indicator_overflow_arhive : Bool;   // Индикатор переполнения архива
      Sum_arhive : Real;   // Сумма всех элементов архива
      R_TRIG_front_impulse : R_TRIG;   // R_TRIG фронта импульса
      Arhive_consumption_TON : IEC_TIMER;
      Moment_consumption_TON : IEC_TIMER;
   END_VAR
BEGIN
   #impulse := "read_discret"(Invert := FALSE, N_module := #impulse_N_module, N_chanel := #impulse_N_chanel);

   (*НАКОПЛЕННЫЙ РАСХОД*)
   #R_TRIG_front_impulse(CLK:=#impulse,
               Q=>#front_impulse);
   //приращение накопленного расхода
   IF #front_impulse THEN
       #accumulated_consumption := #accumulated_consumption + ((#scale_unit)/1000);
   END_IF;
   //сброс накопленного значения счетчика при достичениии max
   IF #accumulated_consumption >= #consumption_max_value THEN
       #correct_consumption := 0.0;
       #apply_correct_consumption := TRUE;
   END_IF;
   //корректировка накопленного расхода
   IF #apply_correct_consumption THEN
       #difference_correct_consumption := #correct_consumption - #accumulated_consumption; //вычисление изменения показаний накопленного расхода
       #Indicator_correct_consumption := TRUE; //взводим индикатор корректировки показаний (для корректировки расхода при архивировании)
       #accumulated_consumption := #correct_consumption;
       #apply_correct_consumption := FALSE;
   END_IF;

   (*МНГОВЕННЫЙ РАСХОД*)
   //вычисление мгновенного расхода
   IF #front_impulse THEN
       #Time_moment_consumption := #Moment_consumption_Timer_ET;
       #Moment_consumption_Timer_IN := FALSE;
       (* мгновенный расход[м3/ч]=(1[ms]/время[ms])*цена импульса[литр]*(60*60*1000)/1000 *)
       #moment_consumption := (3600*(#scale_unit))/UDINT_TO_REAL(T_CONV(#Time_moment_consumption));
   END_IF;
   (*корректировка показаний мгновенного расхода при его снижении*)
   IF #Moment_consumption_Timer_ET > #Time_moment_consumption THEN
       (* мгновенный расход[м3/ч]=(1[ms]/текущее время от предыдущего импульса[ms])*цена импульса[литр]*(60*60*1000)/1000 *)
       #moment_consumption := (3600 * (#scale_unit)) / UDINT_TO_REAL(T_CONV(#Moment_consumption_Timer_ET));
   END_IF;
   #Moment_consumption_TON.TON(IN:=#Moment_consumption_Timer_IN,
                                PT:=#Time_min_consumption,
                                Q=>#Moment_consumption_Timer_Q,
                                ET=>#Moment_consumption_Timer_ET);
   IF #Moment_consumption_Timer_Q THEN
       #moment_consumption := 0;
   END_IF;
   IF NOT #Moment_consumption_Timer_IN THEN
       #Moment_consumption_Timer_IN := TRUE;
   END_IF;

   (*СРЕДНЕСУТОЧНЫЙ РАСХОД*)
   //вычисление среднесуточного расхода (на основе анализа 12 минутных интервалов за последние 30 дней)
   #Arhive_consumption_TON.TON(IN := #Arhive_Timer_IN,
                                     PT := T#12m,
                                     Q => #Arhive_Timer_Q);
   //если произведена корректировка показаний накопленного расхода
   IF #Indicator_correct_consumption THEN
       #accumulated_consumption_T := #accumulated_consumption_T + #difference_correct_consumption; //учитываем в предыдущем расходе корректировку показаний
       #Indicator_correct_consumption := FALSE; //Сбрасываем индикатор корректировки показаний
   END_IF;

   IF #Arhive_Timer_Q THEN
       #Arhive_Timer_IN := FALSE;
       //вычисление расхода за прошедший интервал
       #Current_arhive_cunsumption := #accumulated_consumption - #accumulated_consumption_T;
       #accumulated_consumption_T := #accumulated_consumption;
       //вычисляем сумму всех элементов архива (с учетом возможной перезаписи элемента архива)
       #Sum_arhive := #Sum_arhive - #Arhive_consumption[#marker_arhive]+#Current_arhive_cunsumption;
       //запись расхода за прошедший интервал в архив
       #Arhive_consumption[#marker_arhive] := #Current_arhive_cunsumption;
       //вычисляем среднесуточный расход
       IF NOT #Indicator_overflow_arhive THEN //если архив ещё не заполнен
           (*среднесуточный расход = (120 * сумма элементов массива)/колличествово заполненных элементов массива*)
           #dayly_consumption_average := (120 * #Sum_arhive) / (#marker_arhive+1);
       ELSE    //если архив уже полностью заполнен
           #dayly_consumption_average := #Sum_arhive / 30;
       END_IF;
       //сдвигаем указатель массива
       #marker_arhive := #marker_arhive + 1;
       IF #marker_arhive > 3599 THEN
           #marker_arhive := 0;    //сбрасываем указатель 
           #Indicator_overflow_arhive := TRUE; //взводим индикатор переполнения архива
       END_IF;
   END_IF;
   IF NOT #Arhive_Timer_IN AND NOT #Arhive_Timer_Q THEN
       #Arhive_Timer_IN := TRUE;
   END_IF;
END_FUNCTION_BLOCK

